// TIA Portal V20 export
DATA_BLOCK "ALARM TABLE"   // DB2025
{ S7_Optimized_Access := 'FALSE' }
// stored: AutoNumber false
   VAR
      TAB_01 : Struct
         CNT01 : Int;
         DBX2_0 : Bool;   // 3;AI;Temperatura Apa in Bazin Pompare - Minim Minim;DI;W2;6;O
         DBX2_1 : Bool;   // 3;AI;Temperatura Apa in Bazin Pompare - Minim;DI;W1;6;O
         DBX2_2 : Bool;   // 3;AI;Temperatura Apa in Bazin Pompare - Maxim;DI;A1;6;O
         DBX2_3 : Bool;   // 3;AI;Temperatura Apa in Bazin Pompare - Maxim Maxim;DI;A2;6;O
         DBX2_4 : Bool;   // 3;AI;Temperatura Apa in Bazin Pompare - Senzor Defect;DI;A2;6;M
         DBX2_5 : Bool;   // 3;AI;Temperatura EtilenGlicol Intrare in Racitor - Minim Minim;DI;W1;6;O
         DBX2_6 : Bool;   // 3;AI;Temperatura EtilenGlicol Intrare in Racitor - Minim;DI;W1;6;O
         DBX2_7 : Bool;   // 3;AI;Temperatura EtilenGlicol Intrare in Racitor - Maxim;DI;W1;6;O
         DBX3_0 : Bool;   // 3;AI;Temperatura EtilenGlicol Intrare in Racitor - Maxim Maxim;DI;A1;6;O
         DBX3_1 : Bool;   // 3;AI;Temperatura EtilenGlicol Intrare in Racit. - Senzor Defect;DI;A2;6;M
         DBX3_2 : Bool;   // 3;AI;Temperatura EtilenGlicol Iesire din Racitor - Minim Minim;DI;W1;6;O
         DBX3_3 : Bool;   // 3;AI;Temperatura EtilenGlicol Iesire din Racitor - Minim;DI;W1;6;O
         DBX3_4 : Bool;   // 3;AI;Temperatura EtilenGlicol Iesire din Racitor - Maxim;DI;W1;6;O
         DBX3_5 : Bool;   // 3;AI;Temperatura EtilenGlicol Iesire din Racitor - Maxim Maxim;DI;A1;6;O
         DBX3_6 : Bool;   // 3;AI;Temperatura EtilenGlicol Iesire din Racit. - Senzor Defect;DI;A2;6;M
         DBX3_7 : Bool;   // 3;AI;Temperatura Apa la Iesire din Racitor - Minim Minim;DI;W2;6;O
         DBX4_0 : Bool;   // 3;AI;Temperatura Apa la Iesire din Racitor - Minim;DI;W1;6;O
         DBX4_1 : Bool;   // 3;AI;Temperatura Apa la Iesire din Racitor - Maxim;DI;W2;6;O
         DBX4_2 : Bool;   // 3;AI;Temperatura Apa la Iesire din Racitor - Maxim Maxim;DI;W2;6;O
         DBX4_3 : Bool;   // 3;AI;Temperatura Apa la Iesire din Racitor - Senzor Defect;DI;A2;6;M
         DBX4_4 : Bool;   // 3;AI;Temperatura Apa Alimentare Linia Calire - Minim Minim;DI;A2;3;O
         DBX4_5 : Bool;   // 3;AI;Temperatura Apa Alimentare Linia Calire - Minim;DI;A1;3;M;O
         DBX4_6 : Bool;   // 3;AI;Temperatura Apa Alimentare Linia Calire - Maxim;DI;A1;3;O
         DBX4_7 : Bool;   // 3;AI;Temperatura Apa Alimentare Linia Calire - Maxim Maxim;DI;A2;3;O
         DBX5_0 : Bool;   // 3;AI;Temperatura Apa Alimentare Linia Calire - Senzor Defect;DI;A2;3;M
         DBX5_1 : Bool;   // 3;AI;Temperatura Apa Alimentare Turnuri Racire - Minim Minim;DI;W2;6;O
         DBX5_2 : Bool;   // 3;AI;Temperatura Apa Alimentare Turnuri Racire - Minim;DI;W1;6;O
         DBX5_3 : Bool;   // 3;AI;Temperatura Apa Alimentare Turnuri Racire - Maxim;DI;A1;6;O
         DBX5_4 : Bool;   // 3;AI;Temperatura Apa Alimentare Turnuri Racire - Maxim Maxim;DI;A1;6;O
         DBX5_5 : Bool;   // 3;AI;Temperatura Apa Alimentare Turnuri Racire - Senzor Defect;DI;A2;6;M
         DBX5_6 : Bool;   // 3;AI;Temparatura Apa in Vas Intermediar - Minim Minim;DI;W1;6;O
         DBX5_7 : Bool;   // 3;AI;Temparatura Apa in Vas Intermediar - Minim;DI;W1;6;O
         DBX6_0 : Bool;   // 3;AI;Temparatura Apa in Vas Intermediar - Maxim;DI;A1;6;O
         DBX6_1 : Bool;   // 3;AI;Temparatura Apa in Vas Intermediar - Maxim Maxim;DI;A1;6;O
         DBX6_2 : Bool;   // 3;AI;Temparatura Apa in Vas Intermediar - Senzor Defect;DI;A2;6;M
         DBX6_3 : Bool;   // 3;AI;Presiune Apa Alimentare Linia Calire - Minim Minim;DI;A2;8;O
         DBX6_4 : Bool;   // 3;AI;Presiune Apa Alimentare Linia Calire - Minim;DI;A1;8;O
         DBX6_5 : Bool;   // 3;AI;Presiune Apa Alimentare Linia Calire - Maxim;DI;A1;8;O
         DBX6_6 : Bool;   // 3;AI;Presiune Apa Alimentare Linia Calire - Maxim Maxim;DI;A2;8;O
         DBX6_7 : Bool;   // 3;AI;Presiune Apa Alimentare Linia Calire - Senzor Defect;DI;A2;8;M
         DBX7_0 : Bool;   // 3;AI;Nivel Apa in Bazin Pompare - Minim Minim;DI;A2;6;O;K
         DBX7_1 : Bool;   // 3;AI;Nivel Apa in Bazin Pompare - Minim;DI;A1;6;O
         DBX7_2 : Bool;   // 3;AI;Nivel Apa in Bazin Pompare - Maxim;DI;A1;6;O;K
         DBX7_3 : Bool;   // 3;AI;Nivel Apa in Bazin Pompare - Maxim Maxim;DI;A2;6;O;K
         DBX7_4 : Bool;   // 3;AI;Nivel Apa in Bazin Pompare - Senzor Defect;DI;A2;6;M
         DBX7_5 : Bool;   // 3;AI;Nivel Apa in Basa Generala - Minim Minim;DI;A2;6;O;K
         DBX7_6 : Bool;   // 3;AI;Nivel Apa in Basa Generala - Minim;DI;A1;6;O
         DBX7_7 : Bool;   // 3;AI;Nivel Apa in Basa Generala - Maxim;DI;A1;6;O
         DBX8_0 : Bool;   // 3;AI;Nivel Apa in Basa Generala - Maxim Maxim;DI;A2;6;O
         DBX8_1 : Bool;   // 3;AI;Nivel Apa in Basa Generala - Senzor Defect;DI;A1;6;M;K
         DBX8_2 : Bool;
         DBX8_3 : Bool;
         DBX8_4 : Bool;
         DBX8_5 : Bool;
         DBX8_6 : Bool;
         DBX8_7 : Bool;
         DBX9_0 : Bool;
         DBX9_1 : Bool;
         DBX9_2 : Bool;
         DBX9_3 : Bool;
         DBX9_4 : Bool;
         DBX9_5 : Bool;
         DBX9_6 : Bool;
         DBX9_7 : Bool;
         DBX10_0 : Bool;
         DBX10_1 : Bool;
         DBX10_2 : Bool;
         DBX10_3 : Bool;
         DBX10_4 : Bool;
         DBX10_5 : Bool;
         DBX10_6 : Bool;
         DBX10_7 : Bool;
         DBX11_0 : Bool;
         DBX11_1 : Bool;
         DBX11_2 : Bool;
         DBX11_3 : Bool;
         DBX11_4 : Bool;
         DBX11_5 : Bool;
         DBX11_6 : Bool;
         DBX11_7 : Bool;
         DBX12_0 : Bool;   // 3;AI;Temperatura Teava (pirometru dupa Sutton) - Minim Minim;DI;A2;20;O
         DBX12_1 : Bool;   // 3;AI;Temperatura Teava (pirometru dupa Sutton) - Minim;DI;A1;20;O
         DBX12_2 : Bool;   // 3;AI;Temperatura Teava (pirometru dupa Sutton) - Maxim;DI;A1;20;O
         DBX12_3 : Bool;   // 3;AI;Temperatura Teava (pirometru dupa Sutton) - Maxim Maxim;DI;A2;20;O
         DBX12_4 : Bool;   // 3;AI;Temperatura Teava (pirometru dupa Sutton) - Senzor Defect;DI;A2;20;M
         DBX12_5 : Bool;   // 3;AI;Temperatura Teava (pir. intr. cupt. revenire) - Minim Minim;DI;A1;20;O
         DBX12_6 : Bool;   // 3;AI;Temperatura Teava (pir. intr. cupt. revenire) - Minim;DI;A1;20;O
         DBX12_7 : Bool;   // 3;AI;Temperatura Teava (pir. intr. cupt. revenire) - Maxim;DI;A1;20;O
         DBX13_0 : Bool;   // 3;AI;Temperatura Teava (pir. intr. cupt. revenire) - Maxim Maxim;DI;A2;20;O
         DBX13_1 : Bool;   // 3;AI;Temperatura Teava (pir. intr. cupt. revenire) - Senzor Def.;DI;A2;20;M
         DBX13_2 : Bool;   // 3;AI;Low Low Apa Redox;DI;A2;20;M;O
         DBX13_3 : Bool;
         DBX13_4 : Bool;
         DBX13_5 : Bool;
         DBX13_6 : Bool;
         DBX13_7 : Bool;
         DBX14_0 : Bool;
         DBX14_1 : Bool;
         DBX14_2 : Bool;
         DBX14_3 : Bool;
         DBX14_4 : Bool;
         DBX14_5 : Bool;
         DBX14_6 : Bool;
         DBX14_7 : Bool;
         DBX15_0 : Bool;
         DBX15_1 : Bool;
         DBX15_2 : Bool;
         DBX15_3 : Bool;
         DBX15_4 : Bool;
         DBX15_5 : Bool;
         DBX15_6 : Bool;
         DBX15_7 : Bool;
         DBX16_0 : Bool;
         DBX16_1 : Bool;
         DBX16_2 : Bool;
         DBX16_3 : Bool;
         DBX16_4 : Bool;
         DBX16_5 : Bool;
         DBX16_6 : Bool;
         DBX16_7 : Bool;
         DBX17_0 : Bool;   // 3;AI;Lipsa presiune destunderizator;DI;A2;7;O
         DBX17_1 : Bool;   // 3;AI;Nivel Apa in Bazin Pompare - Minim;DI;A1;7;O
         DBX17_2 : Bool;
         DBX17_3 : Bool;
         DBX17_4 : Bool;
         DBX17_5 : Bool;
         DBX17_6 : Bool;   // 5;ROLLS T6;Problema pirometru intrare cuptor;DI;A1;16;M;O
         DBX17_7 : Bool;   // 4;FIERASTRAU KASTO;Pat racire - Zona Kasto pachete diferite;TK;W2;11;O
         DBX18_0 : Bool;
         DBX18_1 : Bool;
         DBX18_2 : Bool;
         DBX18_3 : Bool;
         DBX18_4 : Bool;
         DBX18_5 : Bool;
         DBX18_6 : Bool;
         DBX18_7 : Bool;
         DBX19_0 : Bool;
         DBX19_1 : Bool;
         DBX19_2 : Bool;
         DBX19_3 : Bool;
         DBX19_4 : Bool;
         DBX19_5 : Bool;
         DBX19_6 : Bool;
         DBX19_7 : Bool;
         DBX20_0 : Bool;
         DBX20_1 : Bool;
         DBX20_2 : Bool;
         DBX20_3 : Bool;
         DBX20_4 : Bool;
         DBX20_5 : Bool;
         DBX20_6 : Bool;
         DBX20_7 : Bool;
         DBX21_0 : Bool;
         DBX21_1 : Bool;
         DBX21_2 : Bool;
         DBX21_3 : Bool;
         DBX21_4 : Bool;
         DBX21_5 : Bool;
         DBX21_6 : Bool;
         DBX21_7 : Bool;
         DBX22_0 : Bool;
         DBX22_1 : Bool;
         DBX22_2 : Bool;
         DBX22_3 : Bool;
         DBX22_4 : Bool;
         DBX22_5 : Bool;
         DBX22_6 : Bool;
         DBX22_7 : Bool;
         DBX23_0 : Bool;
         DBX23_1 : Bool;
         DBX23_2 : Bool;
         DBX23_3 : Bool;
         DBX23_4 : Bool;
         DBX23_5 : Bool;
         DBX23_6 : Bool;
         DBX23_7 : Bool;
         DBX24_0 : Bool;
         DBX24_1 : Bool;
         DBX24_2 : Bool;
         DBX24_3 : Bool;
         DBX24_4 : Bool;
         DBX24_5 : Bool;
         DBX24_6 : Bool;
         DBX24_7 : Bool;
         DBX25_0 : Bool;
         DBX25_1 : Bool;
         DBX25_2 : Bool;
         DBX25_3 : Bool;
         DBX25_4 : Bool;
         DBX25_5 : Bool;
         DBX25_6 : Bool;
         DBX25_7 : Bool;
         DBX26_0 : Bool;
         DBX26_1 : Bool;
         DBX26_2 : Bool;
         DBX26_3 : Bool;
         DBX26_4 : Bool;
         DBX26_5 : Bool;
         DBX26_6 : Bool;
         DBX26_7 : Bool;
         DBX27_0 : Bool;
         DBX27_1 : Bool;
         DBX27_2 : Bool;
         DBX27_3 : Bool;
         DBX27_4 : Bool;
         DBX27_5 : Bool;
         DBX27_6 : Bool;
         DBX27_7 : Bool;
         DBX28_0 : Bool;
         DBX28_1 : Bool;
         DBX28_2 : Bool;
         DBX28_3 : Bool;
         DBX28_4 : Bool;
         DBX28_5 : Bool;
         DBX28_6 : Bool;
         DBX28_7 : Bool;
         DBX29_0 : Bool;
         DBX29_1 : Bool;
         DBX29_2 : Bool;
         DBX29_3 : Bool;
         DBX29_4 : Bool;
         DBX29_5 : Bool;
         DBX29_6 : Bool;
         DBX29_7 : Bool;
         DBX30_0 : Bool;
         DBX30_1 : Bool;
         DBX30_2 : Bool;
         DBX30_3 : Bool;
         DBX30_4 : Bool;
         DBX30_5 : Bool;
         DBX30_6 : Bool;
         DBX30_7 : Bool;
         DBX31_0 : Bool;
         DBX31_1 : Bool;
         DBX31_2 : Bool;
         DBX31_3 : Bool;
         DBX31_4 : Bool;
         DBX31_5 : Bool;
         DBX31_6 : Bool;
         DBX31_7 : Bool;
         DBX32_0 : Bool;   // 1;Gen;Z1:Sistem Oprire de Urgenta T1-A - Declansat;EM;A3;1;M;O;K
         DBX32_1 : Bool;   // 1;Gen;Z2:Sistem Oprire de Urgenta T1-C - Declansat;EM;A3;1;M;O;K
         DBX32_2 : Bool;   // 1;Gen;Z3:Sistem Oprire de Urgenta Apa - Declansat;EM;A3;6;M;O;K
         DBX32_3 : Bool;   // 1;Gen;Z4:Sistem Oprire de Urgenta T3,T4 - Declansat;EM;A3;10;M;O;K
         DBX32_4 : Bool;   // 1;Gen;Z5:Sistem Oprire de Urgenta T5-T6 - Declansat;EM;A3;14;M;O;K
         DBX32_5 : Bool;   // 1;Gen;Z6:Sistem Oprire de Urgenta T1-D - Declansat;EM;A3;16;M;O;K
         DBX32_6 : Bool;   // 1;Gen;Z7:Sistem Oprire de Urgenta T7 - Declansat;EM;A3;21;M;O;K
         DBX32_7 : Bool;   // 1;Gen;Z8:Sistem Oprire de Urgenta T7-A,T7-B,T7-C - Declansat;EM;A3;23;M;O;K
         DBX33_0 : Bool;   // 1;Gen;Lipsa Tensiune Alimentare Intrari Digitale PLC;DI;A1;6;M;K
         DBX33_1 : Bool;   // 1;Gen;Lipsa Tensiune Alimentare Iesiri Digitale PLC;DI;A1;6;M;K
         DBX33_2 : Bool;   // 1;Gen;Lipsa Tensiune Alimentare (220V pt. module ET);DI;A1;6;M;K
         DBX33_3 : Bool;   // 1;Gen;Lipsa Tensiune Alimentare pt. modulele ET-TF1;DI;A1;6;M;K
         DBX33_4 : Bool;   // 1;Gen;Lipsa Tensiune Alimentare pt. modulele ET-TF2;DI;A1;20;M;K
         DBX33_5 : Bool;   // 1;Gen;Lipsa Tensiune Alimentare pt. modulele ET-TF3;DI;A1;6;M;K
         DBX33_6 : Bool;   // 1;Gen;Lipsa Tensiune Alimentare pt. modulele ET-TF4;DI;A1;6;M;K
         DBX33_7 : Bool;   // 1;Gen;Lipsa Tensiune Alimentare pt. modulele ET-LM1;DI;A1;6;M;K
         DBX34_0 : Bool;   // 1;Gen;Lipsa Tensiune Alimentare pt. modulele ET-LM2;DI;A1;6;M;K
         DBX34_1 : Bool;   // 1;Gen;Lipsa Tensiune Alimentare pt. modulele ET-LM4;DI;A1;13;M;K
         DBX34_2 : Bool;   // 1;Gen;Lipsa Tensiune Alimentare pt. modulele ET-LM5;DI;A1;20;M;K
         DBX34_3 : Bool;   // 1;Gen;Lipsa Tensiune Alimentare pt. modulele ET-LM6;DI;A1;27;M;K
         DBX34_4 : Bool;   // 1;Gen;Lipsa Tensiune Alimentare pt. modulele ET-LM7;DI;A1;6;M;K
         DBX34_5 : Bool;   // 1;Gen;Z1:Teava mai lunga de 14m pe T1-A Incarcare imposibila;DI;A3;1;M;O;K
         DBX34_6 : Bool;   // 1;Gen;Lipsa Tensiune Alimentare UPS;DI;W2;6;M
         DBX34_7 : Bool;   // 1;Gen;UPS not OK;DI;W2;6;M
         DBX35_0 : Bool;   // 1;Gen;Lipsa Tensiune Alimentare pt. Electrovalvole (PLC);DI;A1;6;M;K
         DBX35_1 : Bool;   // 1;Gen;Lipsa Tensiune Alimentare pt. Electrovalvole (LM1);DI;A1;6;M;K
         DBX35_2 : Bool;   // 1;Gen;Lipsa Tensiune Alimentare pt. Electrovalvole (LM2);DI;A1;6;M;K
         DBX35_3 : Bool;   // 1;Gen;Lipsa Tensiune Alimentare pt. Electrovalvole (LM4);DI;A1;6;M;K
         DBX35_4 : Bool;   // 1;Gen;Lipsa Tensiune Alimentare pt. Electrovalvole (LM5);DI;A1;6;M;K
         DBX35_5 : Bool;   // 1;Gen;Lipsa Tensiune Alimentare pt. Electrovalvole (LM6);DI;A1;6;M;K
         DBX35_6 : Bool;   // 1;Gen;Lipsa Tensiune Alimentare pt. Electrovalvole (LM7);DI;A1;6;M;K
         DBX35_7 : Bool;   // 1;Gen;Lipsa Tensiune Alimentare pt. Electrovalvole (ET-TF1);DI;A1;6;M;K
         DBX36_0 : Bool;   // 1;Gen;Lipsa Tensiune Alimentare Senzori (LM1);DI;A1;6;M;K
         DBX36_1 : Bool;   // 1;Gen;Lipsa Tensiune Alimentare Senzori(LM2);DI;A1;6;M;K
         DBX36_2 : Bool;   // 1;Gen;Lipsa Tensiune Alimentare Senzori(LM4);DI;A1;6;M;K
         DBX36_3 : Bool;   // 1;Gen;Lipsa Tensiune Alimentare Senzori(LM5);DI;A1;6;M;K
         DBX36_4 : Bool;   // 1;Gen;Lipsa Tensiune Alimentare Senzori(LM6);DI;A1;6;M;K
         DBX36_5 : Bool;   // 1;LM1;Lipsa Tensiune Alimentare Intrari Digitale (LM1);DI;A1;13;M;K
         DBX36_6 : Bool;   // 1;LM1;Lipsa Tensiune Alimentare Iesiri Digitale (LM1);DI;A1;13;M;K
         DBX36_7 : Bool;   // 1;LM1;Lipsa Tensiune Alimentare Modul FM350 (LM1);DI;A1;13;M;K
         DBX37_0 : Bool;
         DBX37_1 : Bool;
         DBX37_2 : Bool;
         DBX37_3 : Bool;   // 1;LM2;Lipsa Tensiune Alimentare Intrari Digitale (LM2);DI;A1;6;M;K
         DBX37_4 : Bool;   // 1;LM2;Lipsa Tensiune Alimentare Iesiri Digitale (LM2);DI;A1;6;M;K
         DBX37_5 : Bool;   // 1;LM2;Lipsa Tensiune Alimentare Modul FM350 (LM2);DI;A1;6;M;K
         DBX37_6 : Bool;
         DBX37_7 : Bool;
         DBX38_0 : Bool;
         DBX38_1 : Bool;   // 1;LM4;Lipsa Tensiune Alimentare Intrari Digitale (LM4);DI;A1;6;M;K
         DBX38_2 : Bool;   // 1;LM4;Lipsa Tensiune Alimentare Iesiri Digitale (LM4);DI;A1;6;M;K
         DBX38_3 : Bool;   // 1;PLC;TimeOut Comunicatie cu PLC-ul de la Cuptorul de Calire;DI;A1;3;M;O;K
         DBX38_4 : Bool;   // 6;PLC;TimeOut Comunicatie cu PLC-ul de la Cuptorul de Revenire;DI;A1;17;M;O;K
         DBX38_5 : Bool;   // 8;PLC;TimeOut Comunicatie cu PLC-ul de la Indreptare Tevi ;DI;A1;22;M;O;K
         DBX38_6 : Bool;
         DBX38_7 : Bool;   // 1;LM5;Lipsa Tensiune Alimentare Intrari Digitale (LM5);DI;A1;20;M;K
         DBX39_0 : Bool;   // 1;LM5;Lipsa Tensiune Alimentare Iesiri Digitale (LM5);DI;A1;20;M;K
         DBX39_1 : Bool;   // 1;LM5;Lipsa Tensiune Alimentare Modul FM350 (LM5);DI;A1;20;M;K
         DBX39_2 : Bool;
         DBX39_3 : Bool;
         DBX39_4 : Bool;
         DBX39_5 : Bool;   // 1;LM6;Lipsa Tensiune Alimentare Intrari Digitale (LM6);DI;A1;27;M;K
         DBX39_6 : Bool;   // 1;LM6;Lipsa Tensiune Alimentare Iesiri Digitale (LM6);DI;A1;27;M;K
         DBX39_7 : Bool;   // 1;LM6;Lipsa Tensiune Alimentare Modul FM350 (LM6);DI;A1;27;M;K
         DBX40_0 : Bool;
         DBX40_1 : Bool;
         DBX40_2 : Bool;
         DBX40_3 : Bool;   // 1;LM7;Lipsa Tensiune Alimentare Intrari Digitale (LM7);DI;A1;27;M;K
         DBX40_4 : Bool;   // 1;LM7;Lipsa Tensiune Alimentare Iesiri Digitale (LM7);DI;A1;27;M;K
         DBX40_5 : Bool;   // 1;LM7;Lipsa Tensiune Alimentare Senzori (LM6);DI;A1;27;M;K
         DBX40_6 : Bool;
         DBX40_7 : Bool;
         DBX41_0 : Bool;   // 1;TF1;Lipsa Tensiune Alimentare Intrari Digitale (TF1);DI;A1;6;M;K
         DBX41_1 : Bool;   // 1;TF1;Lipsa Tensiune Alimentare Iesiri Digitale (TF1);DI;A1;6;M;K
         DBX41_2 : Bool;   // 1;TF1;Lipsa Tensiune Alimentare 380V (TF1);DI;A1;6;M;K
         DBX41_3 : Bool;   // 1;TF1;Lipsa Tensiune Alimentare 220V (TF1);DI;A1;6;M;K
         DBX41_4 : Bool;   // 1;TF1;Disjunctor Termic 220V (TF1) - Declansat;DI;A1;6;M;K
         DBX41_5 : Bool;
         DBX41_6 : Bool;
         DBX41_7 : Bool;   // 1;TF2;Lipsa Tensiune Alimentare Intrari Digitale (TF2);DI;A1;20;M;K
         DBX42_0 : Bool;   // 1;TF2;Lipsa Tensiune Alimentare Iesiri Digitale (TF2);DI;A1;20;M;K
         DBX42_1 : Bool;
         DBX42_2 : Bool;
         DBX42_3 : Bool;   // 1;TF3;Lipsa Tensiune Alimentare Intrari Digitale (TF3);DI;A1;27;M;K
         DBX42_4 : Bool;   // 1;TF3;Lipsa Tensiune Alimentare Iesiri Digitale (TF3);DI;A1;27;M;K
         DBX42_5 : Bool;   // 1;TF3;Lipsa Tensiune Alimentare 380V (TF3);DI;A1;27;M;K
         DBX42_6 : Bool;   // 1;TF3;Lipsa Tensiune Alimentare 220V (TF3);DI;A1;27;M;K
         DBX42_7 : Bool;   // 1;TF3;Disjunctor Termic 220V (TF3) - Declansat;DI;A1;27;M;K
         DBX43_0 : Bool;
         DBX43_1 : Bool;
         DBX43_2 : Bool;   // 1;TF4;Lipsa Tensiune Alimentare Intrari Digitale (TF4);DI;A1;6;M;K
         DBX43_3 : Bool;   // 1;TF4;Lipsa Tensiune Alimentare Senzori (TF4);DI;A1;6;M;K
         DBX43_4 : Bool;
         DBX43_5 : Bool;
         DBX43_6 : Bool;   // 4;Gen;Z4:Sistem Oprire de Urgenta Role RC02 T4 - Declansat;EM;A3;10;M;O;K
         DBX43_7 : Bool;   // 10;Gen;Z27:Sistem Oprire de Urgenta T10 EH01 - Declansat;EM;A3;28;M;O;K
         DBX44_0 : Bool;   // 10;Gen;Z27:Sistem Oprire de Urgenta T10 EH10 - Declansat;EM;A3;28;M;O;K
         DBX44_1 : Bool;   // 10;Gen;Z27:Sistem Oprire de Urgenta T10 EH11 - Declansat;EM;A3;28;M;O;K
         DBX44_2 : Bool;   // 5;Gen;Z15:Sistem Oprire de Urgenta T6 Kasto EH10 - Declansat;EM;A3;15;M;O;K
         DBX44_3 : Bool;   // 9;Gen;Z25:Sistem Oprire de Urgenta T7-C Kasto EH10 - Declansat;EM;A3;25;M;O;K
         DBX44_4 : Bool;
         DBX44_5 : Bool;
         DBX44_6 : Bool;
         DBX44_7 : Bool;
         DBX45_0 : Bool;   // 10;EGH01;Lipsa Tensiune Alimentare 380V (EGH01);DI;A3;28;M;K
         DBX45_1 : Bool;   // 10;EGH01;Lipsa Tensiune Alimentare 230V (EGH01);DI;A2;28;M;K
         DBX45_2 : Bool;   // 10;EGH01;Lipsa Tensiune Alimentare 230V (EGH01);DI;A2;28;M;K
         DBX45_3 : Bool;   // 10;EGH01;Lipsa Tensiune Alimentare 110V (EGH01);DI;A2;28;M;K
         DBX45_4 : Bool;   // 10;EGH01;Lipsa Tensiune Alimentare 24V Convertizoare (EGH01);DI;A2;28;M;K
         DBX45_5 : Bool;   // 10;EGH01;Lipsa Tensiune Alimentare Electrovalve (EGH01);DI;A2;28;M;K
         DBX45_6 : Bool;   // 10;EGH01;Lipsa Tensiune Alimentare MPP1 (EGH01);DI;A2;28;M;K
         DBX45_7 : Bool;   // 10;EGH01;Lipsa Tensiune Alimentare MPP2 (EGH01);DI;A2;28;M;K
         DBX46_0 : Bool;   // 10;EGH01;Lipsa Tensiune Alimentare Kasto 1(EGH01);DI;A3;28;M;K
         DBX46_1 : Bool;   // 10;EH01;Lipsa Tensiune Alimentare ET(EH01);DI;A2;28;M;K
         DBX46_2 : Bool;   // 10;EH01;Lipsa Tensiune Alimentare Intrari Digitale(EH01);DI;A2;28;M;K
         DBX46_3 : Bool;   // 10;EH01;Lipsa Tensiune Alimentare Iesiri Digitale(EH01);DI;A2;28;M;K
         DBX46_4 : Bool;   // 10;EH01;Lipsa Tensiune Alimentare Dispozitive Aux(EH01);DI;A1;28;M;K
         DBX46_5 : Bool;   // 10;EH01;Lipsa Tensiune Alimentare Encodere(EH01);DI;A3;28;M;K
         DBX46_6 : Bool;   // 0;EH01;Disjunctor Alimentare ET - Declansat(EH01);DI;A2;28;M;K
         DBX46_7 : Bool;
         DBX47_0 : Bool;   // 10;ROLLS T10-1;Lipsa Tensiune de Comanda C.Role T10-1;DI;A1;28;M;K
         DBX47_1 : Bool;   // 10;ROLLS T10-1;Probleme Fuzibil C.Role T10-1;DI;A1;28;M;K
         DBX47_2 : Bool;   // 10;ROLLS T10-1;Disj. Termic Mot. C.Role T10-1 - Declansat;DI;A1;28;M;K
         DBX47_3 : Bool;   // 10;ROLLS T10-1;Fuzibil Neinserat C.Role T10-1;DI;A1;28;M;K
         DBX47_4 : Bool;   // 10;ROLLS T10-1;Inverter Mot. C.Role T10-1 - Avarie;DI;A1;28;M;O;K
         DBX47_5 : Bool;   // 10;ROLLS T10-1;Role T10-1 TimeOut Pozitionare Teava;SQ;A1;28;O
         DBX47_6 : Bool;   // 10;ROLLS T10-1;TimeOut Rotire Role C.Role T10-1;DI;A1;28;M;O;K
         DBX47_7 : Bool;   // 10;ROLLS T10-1;TimeOut Cuplare/Decuplare Vent.Mot.C.RoleT10-1;DI;A1;28;M;O
         DBX48_0 : Bool;   // 10;ROLLS T10-1;Disjunctor Th. AlimVent.Mot.C.Role T10-1 Declansat;DI;A1;28;M
         DBX48_1 : Bool;
         DBX48_2 : Bool;
         DBX48_3 : Bool;
         DBX48_4 : Bool;
         DBX48_5 : Bool;
         DBX48_6 : Bool;
         DBX48_7 : Bool;
         DBX49_0 : Bool;
         DBX49_1 : Bool;
         DBX49_2 : Bool;
         DBX49_3 : Bool;
         DBX49_4 : Bool;
         DBX49_5 : Bool;
         DBX49_6 : Bool;   // 3;T3 SERVOVALVE;Lipsa Tensiune Alimentare Servovalva T3;DI;A1;8;M;K
         DBX49_7 : Bool;   // 3;T3 SERVOVALVE;Disjunctor Termic Servovalva - Declansat;DI;A1;8;M;K
         DBX50_0 : Bool;   // 3;PUMP 1;Disjunctor Termic Pompa Apa Nr.1 - Declansat;DI;A1;6;M
         DBX50_1 : Bool;   // 3;PUMP 2;Disjunctor Termic Pompa Apa Nr.2 - Declansat;DI;A1;6;M
         DBX50_2 : Bool;   // 3;PUMP 3;Disjunctor Termic Pompa Apa Nr.3 - Declansat;DI;A1;6;M
         DBX50_3 : Bool;   // 3;PUMP 4;Disjunctor Termic Pompa Apa Nr.4 - Declansat;DI;A1;6;M
         DBX50_4 : Bool;   // 3;PUMP 5;Disjunctor Termic Pompa Apa Nr.5 - Declansat;DI;A1;6;M
         DBX50_5 : Bool;   // 3;PUMP 6;Disjunctor Termic Pompa Apa Nr.6 - Declansat;DI;A1;6;M
         DBX50_6 : Bool;   // 3;PUMP 7;Disjunctor Termic Pompa Apa Nr.7 - Declansat;DI;A1;6;M
         DBX50_7 : Bool;   // 3;PUMP 8;Disjunctor Termic Pompa Apa Nr.8 - Declansat;DI;A1;6;M
         DBX51_0 : Bool;   // 3;PUMP 9;Disjunctor Termic Pompa Apa Nr.9 - Declansat;DI;A1;6;M
         DBX51_1 : Bool;   // 3;PUMP 10;Disjunctor Termic Pompa Apa Nr.10 - Declansat;DI;A1;6;M
         DBX51_2 : Bool;   // 3;PUMP 11;Disjunctor Termic Pompa Apa Nr.11 - Declansat;DI;A1;6;M
         DBX51_3 : Bool;   // 3;TE1;Disjunctor Termic Transportator Elicoidal Nr.1-Declansat;DI;A1;6;M
         DBX51_4 : Bool;   // 3;TE2;Disjunctor Termic Transportator Elicoidal Nr.2-Declansat;DI;A1;6;M
         DBX51_5 : Bool;   // 3;VE1;Disjunctor Termic Ventilator Turn Racire Nr.1-Declansat;DI;A1;6;M
         DBX51_6 : Bool;   // 3;VE2;Disjunctor Termic Ventilator Turn Racire Nr.2-Declansat;DI;A1;6;M
         DBX51_7 : Bool;   // 3;T3 FILTER;Interupator Termic Filtru T3 - Declansat;DI;A1;8;M
         DBX52_0 : Bool;   // 3;PUMP 1;Lipsa Apa in Pompa Apa Nr.1 (senzor curgere);DI;A1;6;M;O
         DBX52_1 : Bool;   // 3;PUMP 2;Lipsa Apa in Pompa Apa Nr.2 (senzor curgere);DI;A1;6;M;O
         DBX52_2 : Bool;   // 3;PUMP 3;Lipsa Apa in Pompa Apa Nr.3 (senzor curgere);DI;A1;6;M;O
         DBX52_3 : Bool;   // 3;PUMP 4;Lipsa Apa in Pompa Apa Nr.4 (senzor curgere);DI;A1;6;M;O
         DBX52_4 : Bool;   // 3;PUMP 5;Lipsa Apa in Pompa Apa Nr.5 (senzor curgere);DI;A1;6;M;O
         DBX52_5 : Bool;   // 3;PUMP 6;Lipsa Apa in Pompa Apa Nr.5R (senzor curgere);DI;A1;6;M;O
         DBX52_6 : Bool;   // 3;PUMP 7;Lipsa Apa in Pompa Apa Nr.7 (senzor curgere);DI;A1;6;M;O
         DBX52_7 : Bool;   // 3;PUMP 8;Lipsa Apa in Pompa Apa Nr.8 (senzor curgere);DI;A1;6;M;O
         DBX53_0 : Bool;   // 3;T3 FILTER;Lipsa Tensiune Alimentare Filtru T3;DI;A1;8;M;K
         DBX53_1 : Bool;   // 3;PUMP 10;Lipsa Apa in Pompa Apa Nr.10 (senzor curgere);DI;A1;6;M;O
         DBX53_2 : Bool;   // 3;BASIN;Lipsa Apa in Bazinul de Pompare;DI;A1;6;O
         DBX53_3 : Bool;   // 3;PUMP 11;Nivel Apa in Casa Pompelor - Minim;DI;A1;6;O
         DBX53_4 : Bool;   // 3;PUMP 11;Nivel Apa in Casa Pompelor - Maxim;DI;A2;6;O;K
         DBX53_5 : Bool;   // 3;BASIN;Nivel Apa in Bazinul de Pompare - Maxim;DI;A2;6;O;K
         DBX53_6 : Bool;   // 3;VESSEL;Nivel Apa in Vasul Intermediar - Minim;DI;A2;6;O;K
         DBX53_7 : Bool;   // 3;T3 FILTER/BEAM;Lipsa Tensiune de Comanda Filtru T3 si Grinda;DI;A2;8;M;K
         DBX54_0 : Bool;   // 3;SCALE;Nivel Apa in Bazinul Tunder - Maxim;DI;A2;6;O;K
         DBX54_1 : Bool;   // 3;SUP;Presiune Apa Scazuta pe Linia de Calire;DI;A1;6;O;K
         DBX54_2 : Bool;   // 3;TOWER;Presiune Apa Scazuta pe Linia de Racire Turnuri;DI;A1;6;O;K
         DBX54_3 : Bool;   // 3;SCP;Temperatura Apa din Schimbatorul de Caldura - Depasita;DI;A2;6;M
         DBX54_4 : Bool;   // 3;BASIN;Temperatura Apa din Bazinul de Pompare - Depasita;DI;A2;6;M;O;K
         DBX54_5 : Bool;   // 3;BASIN;Temperatura Apa din Bazinul de Pompare - Scazuta;DI;A1;6;M;O
         DBX54_6 : Bool;   // 3;BASIN;Avarie Schimbator Caldura (cu EtilenGlicol);DI;A1;6;M;O
         DBX54_7 : Bool;   // 3;DCS;Avarie Sistem DCS;DI;A3;6;M;O;K
         DBX55_0 : Bool;   // 3;F;Avarie Filtru cu Autocuratire;DI;W3;6;O
         DBX55_1 : Bool;   // 3;PUMP 1;TimeOut Cuplare Contactor Pornire Pompa Apa Nr.1;DI;A1;6;M;O;K
         DBX55_2 : Bool;   // 3;PUMP 2;TimeOut Cuplare Contactor Pornire Pompa Apa Nr.2;DI;A1;6;M;O;K
         DBX55_3 : Bool;   // 3;PUMP 3;TimeOut Cuplare Contactor Pornire Pompa Apa Nr.3;DI;A1;6;M;O;K
         DBX55_4 : Bool;   // 3;PUMP 4;TimeOut Cuplare Contactor Pornire Pompa Apa Nr.4;DI;A1;6;M;O;K
         DBX55_5 : Bool;   // 3;PUMP 5;TimeOut Cuplare Contactor Pornire Pompa Apa Nr.5;DI;A1;6;M;O;K
         DBX55_6 : Bool;   // 3;PUMP 5R;TimeOut Cuplare Contactor Pornire Pompa Apa Nr.5R;DI;A1;6;M;O;K
         DBX55_7 : Bool;   // 3;PUMP 7;TimeOut Cuplare Contactor Pornire Pompa Apa Nr.7;DI;A1;6;M;O;K
         DBX56_0 : Bool;   // 3;PUMP 8;TimeOut Cuplare Contactor Pornire Pompa Apa Nr.8;DI;A1;6;M;O;K
         DBX56_1 : Bool;   // 3;PUMP 9;TimeOut Cuplare Contactor Pornire Pompa Apa Nr.9;DI;A1;6;M;O;K
         DBX56_2 : Bool;   // 3;PUMP10;TimeOut Cuplare Contactor Pornire Pompa Apa Nr10;DI;A1;6;M;O;K
         DBX56_3 : Bool;   // 3;PUMP11;TimeOut Cuplare Contactor Pornire Pompa Apa Nr11;DI;A1;6;M;O;K
         DBX56_4 : Bool;   // 3;HELICOIDAL TRANSPORTER 1;TimeOut Transportator Elicoidal Nr.1;DI;A1;6;M;O;K
         DBX56_5 : Bool;   // 3;HELICOIDAL TRANSPORTER 2;TimeOut Transportator Elicoidal Nr.2;DI;A1;6;M;O;K
         DBX56_6 : Bool;   // 3;COOLING TOWER 1;TimeOut Ventilator Turn Racire 1 Viteza Mica;DI;A1;6;M;O;K
         DBX56_7 : Bool;   // 3;COOLING TOWER 1;TimeOut Ventilator Turn Racire 1 Viteza Mare;DI;A1;6;M;O;K
         DBX57_0 : Bool;   // 3;COOLING TOWER 2;TimeOut Ventilator Turn Racire 2 Viteza Mica;DI;A1;6;M;O;K
         DBX57_1 : Bool;   // 3;COOLING TOWER 2;TimeOut Ventilator Turn Racire 2 Viteza Mare;DI;A1;6;M;O;K
         DBX57_2 : Bool;   // 3;T3 FILTER;TimeOut Cuplare/Decuplare Contactor Filtru Inainte;DI;A1;8;M;O;K
         DBX57_3 : Bool;   // 3;T3 FILTER;TimeOut Cuplare/Decuplare Contactor Filtru Inapoi;DI;A1;8;M;O;K
         DBX57_4 : Bool;
         DBX57_5 : Bool;   // 3;T3 SERVOVALVE;Lipsa Tensiune Alimentare Servovalva;DI;A1;8;M;K
         DBX57_6 : Bool;
         DBX57_7 : Bool;
         DBX58_0 : Bool;   // 1;CHAIN T1-A;TimeOut Cuplare Contactor Start Lant T1-A;DI;A1;1;M;O;K
         DBX58_1 : Bool;
         DBX58_2 : Bool;   // 1;CHAIN T1-A;TimeOut Deplasare Lant T1-A in pozitia Pas;DI;A1;1;M;O;K
         DBX58_3 : Bool;   // 1;CHAIN T1-A;Disjunctor Termic Lant T1-A - Declansat;DI;A1;1;M;K
         DBX58_4 : Bool;   // 1;CHAIN T1-A;Sectionator Alimentare Lant T1-A - Decuplat;DI;A1;1;M;K
         DBX58_5 : Bool;   // 1;STOPPER T1-A;Disjunctor Termic Opritor T1-A - Declansat;DI;A1;1;M;K
         DBX58_6 : Bool;   // 1;STOPPER T1-A;Sectionator Alimentare Opritor T1-A - Decuplat;DI;A1;1;M;K
         DBX58_7 : Bool;   // 1;STOPPER T1-A;TimeOut Cuplare Contactor Opritor T1-A;DI;A1;1;M;O;K
         DBX59_0 : Bool;   // 3;T3 FILTER;Lipsa confirmare rotire filtru delta T3;DI;A1;1;M;K
         DBX59_1 : Bool;
         DBX59_2 : Bool;
         DBX59_3 : Bool;
         DBX59_4 : Bool;
         DBX59_5 : Bool;
         DBX59_6 : Bool;
         DBX59_7 : Bool;
         DBX60_0 : Bool;
         DBX60_1 : Bool;
         DBX60_2 : Bool;
         DBX60_3 : Bool;
         DBX60_4 : Bool;
         DBX60_5 : Bool;
         DBX60_6 : Bool;
         DBX60_7 : Bool;
         DBX61_0 : Bool;
         DBX61_1 : Bool;
         DBX61_2 : Bool;
         DBX61_3 : Bool;
         DBX61_4 : Bool;
         DBX61_5 : Bool;
         DBX61_6 : Bool;
         DBX61_7 : Bool;
         DBX62_0 : Bool;   // 1;FLIPPER T1A;Lipsa Tensiune Alimentare Aruncator T1-A;DI;A1;1;M;K
         DBX62_1 : Bool;   // 1;FLIPPER T1A;TimeOut Deplasare Aruncator T1-A in pozitia Sus;DI;A1;1;M;O
         DBX62_2 : Bool;   // 1;FLIPPER T1A;TimeOut Deplasare Aruncator T1-A in pozitia Jos;DI;A1;1;M;O
         DBX62_3 : Bool;   // 1;FLIPPER T1A;Eroare Depozitare Teava pe C.Role T1-A;SQ;A1;1;O
         DBX62_4 : Bool;
         DBX62_5 : Bool;
         DBX62_6 : Bool;
         DBX62_7 : Bool;
         DBX63_0 : Bool;
         DBX63_1 : Bool;
         DBX63_2 : Bool;
         DBX63_3 : Bool;
         DBX63_4 : Bool;
         DBX63_5 : Bool;
         DBX63_6 : Bool;
         DBX63_7 : Bool;
         DBX64_0 : Bool;
         DBX64_1 : Bool;
         DBX64_2 : Bool;
         DBX64_3 : Bool;
         DBX64_4 : Bool;
         DBX64_5 : Bool;
         DBX64_6 : Bool;
         DBX64_7 : Bool;
         DBX65_0 : Bool;
         DBX65_1 : Bool;
         DBX65_2 : Bool;
         DBX65_3 : Bool;
         DBX65_4 : Bool;
         DBX65_5 : Bool;
         DBX65_6 : Bool;
         DBX65_7 : Bool;
         DBX66_0 : Bool;   // 1;ROLLS T1-A;Suma Disjuntoare Termice C.Role T1-A - Declansat;DI;A1;1;M;K
         DBX66_1 : Bool;   // 1;ROLLS T1-A;Sectionator Alim.Inverter C.Role T1-A - Decuplat;DI;A2;1;M;K
         DBX66_2 : Bool;   // 1;ROLLS T1-A;Lipsa Tensiune de Comanda C.Role T1-A;DI;A2;1;M;K
         DBX66_3 : Bool;   // 1;ROLLS T1-A;TimeOut Rotire Role C.Role T1-A;DI;A1;1;M;O;K
         DBX66_4 : Bool;   // 1;ROLLS T1-A;Disj. Termic Rola Nr.1 C.Role T1-A Declansat;DI;W2;1;M
         DBX66_5 : Bool;   // 1;ROLLS T1-A;Disj. Termic Rola Nr.2 C.Role T1-A Declansat;DI;W2;1;M
         DBX66_6 : Bool;   // 1;ROLLS T1-A;Disj. Termic Rola Nr.3 C.Role T1-A Declansat;DI;W2;1;M
         DBX66_7 : Bool;   // 1;ROLLS T1-A;Disj. Termic Rola Nr.4 C.Role T1-A Declansat;DI;W2;1;M
         DBX67_0 : Bool;   // 1;ROLLS T1-A;Disj. Termic Rola Nr.5 C.Role T1-A Declansat;DI;W2;1;M
         DBX67_1 : Bool;   // 1;ROLLS T1-A;Disj. Termic Rola Nr.6 C.Role T1-A Declansat;DI;W2;1;M
         DBX67_2 : Bool;   // 1;ROLLS T1-A;Disj. Termic Rola Nr.7 C.Role T1-A Declansat;DI;W2;1;M
         DBX67_3 : Bool;   // 1;ROLLS T1-A;Disj. Termic Rola Nr.8 C.Role T1-A Declansat;DI;W2;1;M
         DBX67_4 : Bool;   // 1;ROLLS T1-A;TimeOut Cuplare/Decuplare Vent.Mot. C.Role T1-A;DI;W3;1;M
         DBX67_5 : Bool;   // 1;ROLLS T1-A;Disjunctor Th. AlimVent.Mot.C.Role T1A-Declansat;DI;A1;1;M
         DBX67_6 : Bool;
         DBX67_7 : Bool;   // 1;ROLLS T1-A;TimeOut Cuplare Alim.Inverter C.Role T1-A;DI;A1;1;M;O;K
         DBX68_0 : Bool;   // 1;ROLLS T1-A;Suma Disj. Termice Vent.Mot. C.Role T1-A-Declansat;DI;A1;1;M;O
         DBX68_1 : Bool;   // 1;ROLLS T1-A;Inverter Mot. C.Role T1-A - Avarie;DI;A1;1;M;O;K
         DBX68_2 : Bool;   // 1;ROLLS T1-A;Eroare Encoder C.Role T1-A;DI;A1;1;M;O;K
         DBX68_3 : Bool;   // 1;ROLLS T1-A;Role T1-A TimeOut LB Masurare Lungime ON;SQ;A1;1;M;O
         DBX68_4 : Bool;   // 1;ROLLS T1-A;Role T1-A TimeOut LB Masurare Lungime OFF;SQ;A1;1;M;O
         DBX68_5 : Bool;
         DBX68_6 : Bool;
         DBX68_7 : Bool;
         DBX69_0 : Bool;
         DBX69_1 : Bool;
         DBX69_2 : Bool;
         DBX69_3 : Bool;
         DBX69_4 : Bool;
         DBX69_5 : Bool;
         DBX69_6 : Bool;
         DBX69_7 : Bool;
         DBX70_0 : Bool;   // 1;CHAIN T1-C;TimeOut Cuplare/Decuplare Contactor Lant T1-C;DI;A1;2;M;O;K
         DBX70_1 : Bool;
         DBX70_2 : Bool;   // 1;CHAIN T1-C;TimeOut Deplasare Lant T1-C in pozitia Pas;DI;A1;2;M;O;K
         DBX70_3 : Bool;   // 1;CHAIN T1-C;Disjunctor Termic Lant T1-C - Declansat;DI;A1;2;M;K
         DBX70_4 : Bool;   // 1;CHAIN T1-C;Sectionator Alimentare Lant T1-C - Decuplat;DI;A1;2;M;K
         DBX70_5 : Bool;   // 1;STOPPER T1-C;Disjunctor Termic Opritor T1-C - Declansat;DI;A1;2;M;K
         DBX70_6 : Bool;   // 1;STOPPER T1-C;Sectionator Alimentare Opritor T1-C - Decuplat;DI;A1;2;M;K
         DBX70_7 : Bool;   // 1;STOPPER T1-C;TimeOut Cuplare Contactor Opritor T1-C;DI;A1;2;M;O;K
         DBX71_0 : Bool;
         DBX71_1 : Bool;
         DBX71_2 : Bool;
         DBX71_3 : Bool;
         DBX71_4 : Bool;
         DBX71_5 : Bool;
         DBX71_6 : Bool;
         DBX71_7 : Bool;
         DBX72_0 : Bool;
         DBX72_1 : Bool;
         DBX72_2 : Bool;
         DBX72_3 : Bool;
         DBX72_4 : Bool;
         DBX72_5 : Bool;
         DBX72_6 : Bool;
         DBX72_7 : Bool;
         DBX73_0 : Bool;
         DBX73_1 : Bool;
         DBX73_2 : Bool;
         DBX73_3 : Bool;
         DBX73_4 : Bool;
         DBX73_5 : Bool;
         DBX73_6 : Bool;
         DBX73_7 : Bool;
         DBX74_0 : Bool;   // 1;FLIPPER T1C;Lipsa Tensiune Alimentare Aruncator T1-C;DI;A1;2;M;K
         DBX74_1 : Bool;   // 1;FLIPPER T1C;TimeOut Deplasare Aruncator T1-C in pozitia Sus;DI;A1;2;M;O
         DBX74_2 : Bool;   // 1;FLIPPER T1C;TimeOut Deplasare Aruncator T1-C in pozitia Jos;DI;A1;2;M;O
         DBX74_3 : Bool;   // 1;FLIPPER T1C;Eroare Depozitare Teava pe C.Role;SQ;A1;2;O
         DBX74_4 : Bool;
         DBX74_5 : Bool;
         DBX74_6 : Bool;
         DBX74_7 : Bool;
         DBX75_0 : Bool;
         DBX75_1 : Bool;
         DBX75_2 : Bool;
         DBX75_3 : Bool;
         DBX75_4 : Bool;
         DBX75_5 : Bool;
         DBX75_6 : Bool;
         DBX75_7 : Bool;
         DBX76_0 : Bool;
         DBX76_1 : Bool;
         DBX76_2 : Bool;
         DBX76_3 : Bool;
         DBX76_4 : Bool;
         DBX76_5 : Bool;
         DBX76_6 : Bool;
         DBX76_7 : Bool;
         DBX77_0 : Bool;
         DBX77_1 : Bool;
         DBX77_2 : Bool;
         DBX77_3 : Bool;
         DBX77_4 : Bool;
         DBX77_5 : Bool;
         DBX77_6 : Bool;
         DBX77_7 : Bool;
         DBX78_0 : Bool;   // 1;ROLLS T1-C;Suma Disjuntoare Termice C.Role T1-C Declansat;DI;A1;2;M;K
         DBX78_1 : Bool;   // 1;ROLLS T1-C;Sectionator Alim.Inverter C.Role T1-C Decuplat;DI;A2;2;M;K
         DBX78_2 : Bool;   // 1;ROLLS T1-C;Lipsa Tensiune de Comanda C.Role T1-C;DI;A2;2;M;K
         DBX78_3 : Bool;   // 1;ROLLS T1-C;TimeOut Rotire Role C.Role T1-C;DI;A1;2;M;O;K
         DBX78_4 : Bool;   // 1;ROLLS T1-C;Disjunctor Termic Rola Nr.1 C.Role T1-C Declansat;DI;W2;2;M
         DBX78_5 : Bool;   // 1;ROLLS T1-C;Disjunctor Termic Rola Nr.2 C.Role T1-C Declansat;DI;W2;2;M
         DBX78_6 : Bool;   // 1;ROLLS T1-C;Disjunctor Termic Rola Nr.3 C.Role T1-C Declansat;DI;W2;2;M
         DBX78_7 : Bool;   // 1;ROLLS T1-C;Disjunctor Termic Rola Nr.4 C.Role T1-C Declansat;DI;W2;2;M
         DBX79_0 : Bool;   // 1;ROLLS T1-C;Disjunctor Termic Rola Nr.5 C.Role T1-C Declansat;DI;W2;2;M
         DBX79_1 : Bool;   // 1;ROLLS T1-C;Disjunctor Termic Rola Nr.6 C.Role T1-C Declansat;DI;W2;2;M
         DBX79_2 : Bool;   // 1;ROLLS T1-C;Disjunctor Termic Rola Nr.7 C.Role T1-C Declansat;DI;W2;2;M
         DBX79_3 : Bool;   // 1;ROLLS T1-C;Disjunctor Termic Rola Nr.8 C.Role T1-C Declansat;DI;W2;2;M
         DBX79_4 : Bool;   // 1;ROLLS T1-C;Disjunctor Termic Rola Nr.9 C.Role T1-C Declansat;DI;W2;2;M
         DBX79_5 : Bool;   // 1;ROLLS T1-C;Disjunctor Termic Rola Nr10 C.Role T1-C Declansat;DI;W2;2;M
         DBX79_6 : Bool;   // 1;ROLLS T1-C;Disjunctor Termic Rola Nr11 C.Role T1-C Declansat;DI;W2;2;M
         DBX79_7 : Bool;   // 1;ROLLS T1-C;Disjunctor Termic Rola Nr12 C.Role T1-C Declansat;DI;W2;2;M
         DBX80_0 : Bool;   // 1;ROLLS T1-C;Disjunctor Termic Rola Nr13 C.Role T1-C Declansat;DI;W2;2;M
         DBX80_1 : Bool;   // 1;ROLLS T1-C;Eroare Encoder C.Role T1-C;DI;A2;2;M;O;K
         DBX80_2 : Bool;   // 1;ROLLS T1-C;Disjunctor Termic Vent.Mot C.Role T1C Declansat;DI;A1;2;M
         DBX80_3 : Bool;   // 1;ROLLS T1-C;TimeOut Cuplare/Decuplare Vent.Mot C.Role T1-C;DI;A1;2;M;O
         DBX80_4 : Bool;   // 1;ROLLS T1-C;TimeOut Cuplare Alim.InverterC.Role T1-C;DI;A1;2;M;O;K
         DBX80_5 : Bool;   // 1;ROLLS T1-C;Inverter Mot. C.Role T1-C Avarie;DI;A1;2;M;O;K
         DBX80_6 : Bool;   // 1;ROLLS T1-C;Role T1-C TimeOut LB Masurare Lungime ON;SQ;A1;2;M;O
         DBX80_7 : Bool;   // 1;ROLLS T1-C;Role T1-C TimeOut LB Masurare Lungime OFF;SQ;A1;2;M;O
         DBX81_0 : Bool;
         DBX81_1 : Bool;
         DBX81_2 : Bool;
         DBX81_3 : Bool;
         DBX81_4 : Bool;
         DBX81_5 : Bool;
         DBX81_6 : Bool;
         DBX81_7 : Bool;
         DBX82_0 : Bool;   // 10;EXCENTRIC T10;Lipsa Tensiune de Comanda Excentric T10;DI;A1;28;M;K
         DBX82_1 : Bool;   // 10;EXCENTRIC T10;Probleme Fuzibil Excentric T10;DI;A1;28;M;K
         DBX82_2 : Bool;   // 10;EXCENTRIC T10;Disjunctor Termic Mot. Excentric T10 - Declansat;DI;A1;28;M;K
         DBX82_3 : Bool;   // 10;EXCENTRIC T10;Fuzibil Neinserat Excentric T10;DI;A1;28;M;K
         DBX82_4 : Bool;   // 10;EXCENTRIC T10;Inverter Mot. Excentric T10 - Avarie;DI;A1;28;M;O;K
         DBX82_5 : Bool;   // 10;EXCENTRIC T10;Disjunctor Frana Excentric T10 - Declansat;DI;A1;28;M;K
         DBX82_6 : Bool;   // 10;EXCENTRIC T10;Disjunctor Th.AlimVent.Mot.ExcentricT10 Declansat;DI;A1;28;M
         DBX82_7 : Bool;   // 10;EXCENTRIC T10;TimeOut Deplasare Inainte/Inapoi Excentric T10;DI;A1;28;M;O;K
         DBX83_0 : Bool;   // 10;EXCENTRIC T10;TimeOut Deplasare Excentric T10 in Pozitie;DI;A1;28;M;O;K
         DBX83_1 : Bool;   // 10;EXCENTRIC T10;Comunicatie Pierduta Encoder T10;DI;A2;28;M;O;K
         DBX83_2 : Bool;   // 10;EXCENTRIC T10;Senzor Home nedetectat sau defect;DI;A1;28;M;O;K
         DBX83_3 : Bool;   // 10;EXCENTRIC T10;TimeOut Cuplare/Decuplare Vent.Mot ExcentricT10;DI;A1;28;M;O
         DBX83_4 : Bool;   // 10;EXCENTRIC T10;Eroare Depozitare Teava pe Pat Racire T10;SQ;A1;28;O
         DBX83_5 : Bool;   // 10;EXCENTRIC T10;TimeOut Cuplare/Decuplare Frana Excentric T10;DI;A1;28;M;O;K
         DBX83_6 : Bool;
         DBX83_7 : Bool;
         DBX84_0 : Bool;   // 10;CHAIN T10;Lipsa Tensiune de Comanda Lant T10;DI;A1;28;M;K
         DBX84_1 : Bool;   // 10;CHAIN T10;Probleme Fuzibil Lant T10;DI;A1;28;M;K
         DBX84_2 : Bool;   // 10;CHAIN T10;Disjunctor Termic Mot. Lant T10 - Declansat;DI;A1;28;M;K
         DBX84_3 : Bool;   // 10;CHAIN T10;Fuzibil Neinserat Lant T10;DI;A1;28;M;K
         DBX84_4 : Bool;   // 10;CHAIN T10;Inverter Mot. Lant T10 - Avarie;DI;A1;28;M;O;K
         DBX84_5 : Bool;   // 10;CHAIN T10;Disjunctor Frana Lant T10 - Declansat;DI;A1;28;M;O;K
         DBX84_6 : Bool;   // 10;CHAIN T10;Disjunctor Termic Alim. Vent.Mot. Lant T10 - Declansat;DI;A1;28;M
         DBX84_7 : Bool;   // 10;CHAIN T10;Senzor Incetinire T10 - Avarie(blocat pe "activat");DI;A1;28;M;O;K
         DBX85_0 : Bool;   // 10;CHAIN T10;TimeOut Deplasare Lant T10;DI;A1;28;M;O;K
         DBX85_1 : Bool;   // 10;CHAIN T10;Comunicatie Pierduta Encoder Lant T10;DI;A2;28;M;O;K
         DBX85_2 : Bool;   // 10;CHAIN T10;Senzor home nedetectat sau defect;DI;A1;28;M;O;K
         DBX85_3 : Bool;   // 10;CHAIN T10;TimeOut Cuplare/Decuplare Alim.Inv. Lant T10;DI;A1;28;M;O;K
         DBX85_4 : Bool;   // 10;CHAIN T10;TimeOut Deplasare Lant T10 in pozitia Pas;DI;A1;28;M;O;K
         DBX85_5 : Bool;   // 10;CHAIN T10;Eroare Depozitare Teava pe Opritor dupa Lant T10;DI;A1;28;O
         DBX85_6 : Bool;   // 10;CHAIN T10;TimeOut Cuplare/Decuplare Frana Lant T10;DI;A1;28;M;O;K
         DBX85_7 : Bool;
         DBX86_0 : Bool;   // 10;CHAIN T10 SPIN;Lipsa Tensiune de Comanda Rostogolire T10;DI;A2;28;M;K
         DBX86_1 : Bool;   // 10;CHAIN T10 SPIN;Probleme Fuzibil Rostogolire T10;DI;A1;28;M;K
         DBX86_2 : Bool;   // 10;CHAIN T10 SPIN;Disjunctor Lant Rostogolire T10;DI;A1;28;M;K
         DBX86_3 : Bool;   // 10;CHAIN T10 SPIN;Fuzibil Neinserat Rostogolire T10;DI;A1;28;M;K
         DBX86_4 : Bool;   // 10;CHAIN T10 SPIN;Inverter Mot. LantRost. T10 - Avarie;DI;A1;28;M;O;K
         DBX86_5 : Bool;   // 10;CHAIN T10 SPIN;Disjunctor Frana Rostogolire T10-Declansat;DI;A1;28;M;O;K
         DBX86_6 : Bool;   // 10;CHAIN T10 SPIN;Disj. Th. AlimVent.Mot.Lant Rost T10 Declansa;DI;A1;28;M;O;K
         DBX86_7 : Bool;   // 10;CHAIN T10 SPIN;TimeOut Deplasare LantRost. T10;DI;A1;28;M;O;K
         DBX87_0 : Bool;   // 10;CHAIN T10 SPIN;TimeOut Cuplare/Decuplare Vent.Mot LantRost;DI;A1;28;M;O
         DBX87_1 : Bool;
         DBX87_2 : Bool;
         DBX87_3 : Bool;
         DBX87_4 : Bool;
         DBX87_5 : Bool;   // 10;STOPPER T10;TimeOut Deplasare Opritor T10 in pozitia Sus;DI;A1;28;O
         DBX87_6 : Bool;   // 10;STOPPER T10;TimeOut Deplasare Opritor T10 in pozitia Jos;DI;A1;28;O
         DBX87_7 : Bool;   // 10;STOPPER T10;Eroare Depozitare Teava pe C.Role T10-2;SQ;A1;28;O
         DBX88_0 : Bool;
         DBX88_1 : Bool;
         DBX88_2 : Bool;
         DBX88_3 : Bool;
         DBX88_4 : Bool;
         DBX88_5 : Bool;
         DBX88_6 : Bool;
         DBX88_7 : Bool;
         DBX89_0 : Bool;
         DBX89_1 : Bool;
         DBX89_2 : Bool;
         DBX89_3 : Bool;
         DBX89_4 : Bool;   // 4;ROLLS T3;Coliziune teava in Calitor;DI;A3;8;M;O
         DBX89_5 : Bool;   // 4;ROLLS T3;Disjunctor Termic Vent.Mot. C.Role T3 - Declansat;DI;A1;8;M
         DBX89_6 : Bool;   // 4;ROLLS T3;Inverter Mot. C.Role T3 - Avarie;DI;A1;8;M;O;K
         DBX89_7 : Bool;   // 4;ROLLS T3;TimeOut Cuplare/Decuplare Vent.Mot. C.Role T3;DI;A1;8;M;O
         DBX90_0 : Bool;   // 4;ROLLS T3;Lipsa Tensiune de Comanda C.Role T3;DI;A1;8;M;K
         DBX90_1 : Bool;   // 4;ROLLS T3;Sectionator Alim.Inverter Mot. C.Role T3-Decuplat;DI;A1;8;M;K
         DBX90_2 : Bool;   // 4;ROLLS T3;Suma Disjunctoare Termice Mot.C.Role T3-Declansat;DI;A1;8;M;K
         DBX90_3 : Bool;   // 4;ROLLS T3;Disjunctor Termic Rola Nr.1 C.Role T3 Declansat;DI;W2;8;M
         DBX90_4 : Bool;   // 4;ROLLS T3;Disjunctor Termic Rola Nr.2 C.Role T3 Declansat;DI;W2;8;M
         DBX90_5 : Bool;   // 4;ROLLS T3;Disjunctor Termic Rola Nr.3 C.Role T3 Declansat;DI;W2;8;M
         DBX90_6 : Bool;   // 4;ROLLS T3;Disjunctor Termic Rola Nr.4 C.Role T3 Declansat;DI;W2;8;M
         DBX90_7 : Bool;   // 4;ROLLS T3;Disjunctor Termic Rola Nr.5 C.Role T3 Declansat;DI;W2;8;M
         DBX91_0 : Bool;   // 4;ROLLS T3;TimeOut Rotire Role C.Role T3;DI;A1;8;M;O;K
         DBX91_1 : Bool;   // 4;ROLLS T3;TimeOut Cuplare/Decuplare Alim.Inv. C.Role T3;DI;A1;8;M;O;K
         DBX91_2 : Bool;   // 4;DEZTUNDERIZATOR;Disjunctor Term. Deztunderizator-Declansat;DI;A2;7;M;O;K
         DBX91_3 : Bool;   // 4;DEZTUNDERIZATOR;Sectionator Alim. Deztunderizator-Decuplat;DI;A1;7;M;K
         DBX91_4 : Bool;   // 4;DEZTUNDERIZATOR;SoftStarter SIKO Destunderizator - Avarie;DI;A2;7;M;O;K
         DBX91_5 : Bool;
         DBX91_6 : Bool;   // 4;DEZTUNDERIZATOR;Lipsa Tensiune de Comanda Deztunderizator;DI;A1;7;M;O;K
         DBX91_7 : Bool;   // 4;HEADHARD1;Disjunctor Termic Mot. Cap Calire Nr.1-Declansat;DI;A1;8;M;K
         DBX92_0 : Bool;   // 4;HEADHARD1;Disj. Termic Alim. Mot. Cap Calire Nr.1-Decuplat;DI;A1;8;M;K
         DBX92_1 : Bool;   // 4;HEADHARD1;TimeOut Deplasare Cap Calire Nr.1;DI;A1;8;M;O
         DBX92_2 : Bool;   // 4;DEZTUNDERIZATOR;Lipsa Tensiune Alimentare 24V Deztunder;DI;A1;8;M;K
         DBX92_3 : Bool;   // 4;HEADHARD2;Disjunctor Termic Mot. Cap Calire Nr.2-Declansat;DI;A1;8;M;K
         DBX92_4 : Bool;   // 4;HEADHARD2;Disj. Termic Alim. Mot. Cap Calire Nr.2-Decuplat;DI;A1;8;M;K
         DBX92_5 : Bool;   // 4;HEADHARD2;TimeOut Deplasare Cap Calire Nr.2;DI;A1;8;M;O
         DBX92_6 : Bool;
         DBX92_7 : Bool;   // 4;HEADHARD3;Disjunctor Termic Mot. Cap Calire Nr.3-Declansat;DI;A1;8;M;K
         DBX93_0 : Bool;   // 4;HEADHARD3;Disj. Termic Alim. Mot. Cap Calire Nr.3-Decuplat;DI;A1;8;M;K
         DBX93_1 : Bool;   // 4;HEADHARD3;TimeOut Deplasare Cap Calire Nr.3;DI;A1;8;M;O
         DBX93_2 : Bool;
         DBX93_3 : Bool;   // 4;BEAM;Disjunctor Termic Mot. Grinda - Declansat;DI;A1;8;M;K
         DBX93_4 : Bool;   // 4;BEAM;Disjunctor Termic Alim. Mot. Grinda - Decuplat;DI;A1;8;M;K
         DBX93_5 : Bool;   // 4;BEAM;BEAN:TimeOut Deplasare Grinda;DI;A1;8;M;O
         DBX93_6 : Bool;   // 4;BEAM;Lipsa Tensiune Comanda Grinda/Deztunderizator;DI;A1;8;M;K
         DBX93_7 : Bool;   // 4;ROLLS T3;Suma Disj. Termice Vent.Mot. C.Role T3 - Declansat;DI;A1;8;M
         DBX94_0 : Bool;   // 4;ROLLS T4-1;Suma Disj. Termice Mot. C.Role T4-1 - Declansat;DI;A1;10;M;K
         DBX94_1 : Bool;   // 4;ROLLS T4-1;Sectionator Alim.Inv. Mot. C.Role T4-1-Decuplat;DI;A1;10;M;K
         DBX94_2 : Bool;   // 4;ROLLS T4-1;Lipsa Tensiune de Comanda C.Role T4-1;DI;A1;10;M;K
         DBX94_3 : Bool;   // 4;ROLLS T4-1;TimeOut Rotire Role C.Role T4-1;DI;A1;10;M;O;K
         DBX94_4 : Bool;   // 4;ROLLS T4-1;Disj. Termic Rola Nr.1 C.Role T4-1 Declansat;DI;W2;10;M
         DBX94_5 : Bool;   // 4;ROLLS T4-1;Disj. Termic Rola Nr.2 C.Role T4-1 Declansat;DI;W2;10;M
         DBX94_6 : Bool;   // 4;ROLLS T4-1;Disj. Termic Rola Nr.3 C.Role T4-1 Declansat;DI;W2;10;M
         DBX94_7 : Bool;   // 4;ROLLS T4-1;Disj. Termic Rola Nr.4 C.Role T4-1 Declansat;DI;W2;10;M
         DBX95_0 : Bool;   // 4;ROLLS T4-1;Disj. Termic Rola Nr.5 C.Role T4-1 Declansat;DI;W2;10;M
         DBX95_1 : Bool;   // 4;ROLLS T4-1;Disj. Termic Rola Nr.6 C.Role T4-1 Declansat;DI;W2;10;M
         DBX95_2 : Bool;   // 4;ROLLS T4-1;Disj. Termic Rola Nr.7 C.Role T4-1 Declansat;DI;W2;10;M
         DBX95_3 : Bool;   // 4;ROLLS T4-1;Disj. Termic Rola Nr.8 C.Role T4-1 Declansat;DI;W2;10;M
         DBX95_4 : Bool;   // 4;ROLLS T4-1;Disj. Termic Rola Nr.9 C.Role T4-1 Declansat;DI;W2;10;M
         DBX95_5 : Bool;   // 4;ROLLS T4-1;Disjunctor Th. AlimVent.Mot.C.Role T4-1 Declansat;DI;A1;10;M
         DBX95_6 : Bool;   // 4;ROLLS T4-1;Role T4-1 TimeOut Pozitionare Teava;SQ;A1;10;O
         DBX95_7 : Bool;
         DBX96_0 : Bool;
         DBX96_1 : Bool;
         DBX96_2 : Bool;   // 4;ROLLS T4-1;Suma Disj. Th. Vent.Mot. C.Role T4-1-Declansat;DI;A1;10;M
         DBX96_3 : Bool;   // 4;ROLLS T4-1;TimeOut Cuplare/Decuplare Vent.Mot.C.Role T4-1;DI;A1;10;M;O
         DBX96_4 : Bool;   // 4;ROLLS T4-1;TimeOut Cuplare Alim.Inv. C.Role T4-1;DI;A1;10;M;O;K
         DBX96_5 : Bool;   // 4;ROLLS T4-1;Inverter Mot. C.Role T4-1 - Avarie;DI;A1;10;M;O;K
         DBX96_6 : Bool;
         DBX96_7 : Bool;
         DBX97_0 : Bool;   // 4;DEZTUNDERIZATOR;Disjunctor Termic Pompa 9.1 - Declansat;DI;A1;7;M;K
         DBX97_1 : Bool;   // 4;DEZTUNDERIZATOR;Disjunctor Termic Pompa 9.2 - Declansat;DI;A1;7;M;K
         DBX97_2 : Bool;   // 4;DEZTUNDERIZATOR;Lipsa confirm. cuplare contactor Pompa 9.1;DI;A1;7;M;K
         DBX97_3 : Bool;   // 4;DEZTUNDERIZATOR;Lipsa confirm. cuplare contactor Pompa 9.2;DI;A1;7;M;K
         DBX97_4 : Bool;   // 4;DEZTUNDERIZATOR;Sistem Oprire de Urgenta Hammelman-Declansat;EM;A1;7;M;O;K
         DBX97_5 : Bool;   // 4;DEZTUNDERIZATOR;Alarma generala Unitate Hammelmann;DI;A1;7;M;O;K
         DBX97_6 : Bool;   // 4;DEZTUNDERIZATOR;Lipsa confirm robinet izolare deschis 100bar;DI;A1;7;M;O;K
         DBX97_7 : Bool;   // 4;DEZTUNDERIZATOR;Lipsa confirm robinet izolare deschis 180bar;DI;A1;7;M;O;K
         DBX98_0 : Bool;   // 4;EXCENTRIC T4;TimeOut Deplasare Inainte Excentric T4;DI;A1;10;M;O;K
         DBX98_1 : Bool;   // 4;EXCENTRIC T4;TimeOut Deplasare Inapoi Excentric T4;DI;A1;10;M;O;K
         DBX98_2 : Bool;   // 4;EXCENTRIC T4;TimeOut Deplasare Excentric T4 in Pozitie;DI;A1;10;M;O;K
         DBX98_3 : Bool;   // 4;EXCENTRIC T4;Disjunctor Termic Mot. Excentric T4-Declansat;DI;A1;10;M;K
         DBX98_4 : Bool;   // 4;EXCENTRIC T4;Alim. SoftStarter SIKO Excentric T4-Decuplat;DI;A1;10;M;K
         DBX98_5 : Bool;   // 4;EXCENTRIC T4;Alim. Frana Mot. Excentric T4 - Decuplat;DI;A1;10;M;K
         DBX98_6 : Bool;   // 4;EXCENTRIC T4;Lipsa Tensiune de Comanda Excentric T4;DI;A1;10;M;K
         DBX98_7 : Bool;   // 4;EXCENTRIC T4;SoftStarter SIKO Excentric T4 - Avarie;DI;A1;10;M;O;K
         DBX99_0 : Bool;   // 4;EXCENTRIC T4;Eroare Depozitare Teava pe Pat Racire T4;SQ;A1;10;O
         DBX99_1 : Bool;
         DBX99_2 : Bool;
         DBX99_3 : Bool;
         DBX99_4 : Bool;
         DBX99_5 : Bool;
         DBX99_6 : Bool;
         DBX99_7 : Bool;
         DBX100_0 : Bool;   // 4;DEZTUNDERIZATOR;Presiune prea mica inainte de P. Hammelmann;DI;A1;7;O;K
         DBX100_1 : Bool;   // 4;DEZTUNDERIZATOR;Presiune prea mare dupa unit joasa pres.;DI;A1;7;O;K
         DBX100_2 : Bool;   // 4;DEZTUNDERIZATOR;Lipsa confirmare curgere pe alimentare;DI;A1;7;M;O;K
         DBX100_3 : Bool;
         DBX100_4 : Bool;
         DBX100_5 : Bool;
         DBX100_6 : Bool;
         DBX100_7 : Bool;
         DBX101_0 : Bool;
         DBX101_1 : Bool;
         DBX101_2 : Bool;
         DBX101_3 : Bool;
         DBX101_4 : Bool;
         DBX101_5 : Bool;
         DBX101_6 : Bool;
         DBX101_7 : Bool;
         DBX102_0 : Bool;   // 4;CHAIN T4;Stop Permisie Cuplare Lant T4 - Actionat;DI;A1;10;M;O;K
         DBX102_1 : Bool;   // 4;CHAIN T4;TimeOut Cuplare/Decuplare Alim.Inv. Lant T4;DI;A1;10;M;O;K
         DBX102_2 : Bool;   // 4;CHAIN T4;Lipsa Tensiune de Comanda Lant T4;DI;A1;10;M;K
         DBX102_3 : Bool;   // 4;CHAIN T4;Sectionator Alim.Inv. Mot. Lant T4 - Decuplat;DI;A1;10;M;K
         DBX102_4 : Bool;   // 4;CHAIN T4;Alim. Frana Mot. Lant T4 - Decuplat;DI;A1;10;M;K
         DBX102_5 : Bool;   // 4;CHAIN T4;Inverter Mot. Lant T4 - Avarie;DI;A1;10;M;O;K
         DBX102_6 : Bool;   // 4;CHAIN T4 SPIN;TimeOut Cuplare/Decupl. Alim.Inv.LantRost. T4;DI;A1;10;M;O;K
         DBX102_7 : Bool;   // 4;CHAIN T4 SPIN;Sectionator Alim.Inv Mot.LantRost T4-Decuplat;DI;A1;10;M;K
         DBX103_0 : Bool;   // 4;CHAIN T4 SPIN;Disjunctor Termic Mot. LantRost. T4-Declansat;DI;A1;10;M;K
         DBX103_1 : Bool;   // 4;CHAIN T4;TimeOut Deplasare Lant T4 in pozitia Pas;DI;A1;10;M;O;K
         DBX103_2 : Bool;   // 4;CHAIN T4 SPIN;Inverter Mot. LantRost. T4 - Avarie;DI;A1;10;M;O;K
         DBX103_3 : Bool;   // 4;CHAIN T4 SPIN;Stop Permisie Cuplare LantRost. T4 - Actionat;DI;A1;10;M;O;K
         DBX103_4 : Bool;   // 4;CHAIN T4;TimeOut Deplasare Lant T4;DI;A1;10;M;O;K
         DBX103_5 : Bool;   // 4;CHAIN T4;TimeOut Cuplare/Decuplare Frana Lant T4;DI;A1;10;M;O;K
         DBX103_6 : Bool;   // 4;CHAIN T4 SPIN;TimeOut Deplasare LantRost. T4;DI;A1;10;M;O;K
         DBX103_7 : Bool;   // 4;CHAIN T4;Disjunctor Termic Alim. Vent.Mot. Lant T4-Declansat;DI;A1;10;M
         DBX104_0 : Bool;
         DBX104_1 : Bool;
         DBX104_2 : Bool;
         DBX104_3 : Bool;   // 4;CHAIN T4;Eroare Depozitare Teava pe Opritor dupa Lant T4;DI;A1;10;O
         DBX104_4 : Bool;   // 4;CHAIN T4;Senzor Incetinire T4 - Avarie(blocat pe "activat");DI;A1;10;M;O;K
         DBX104_5 : Bool;
         DBX104_6 : Bool;
         DBX104_7 : Bool;
         DBX105_0 : Bool;
         DBX105_1 : Bool;
         DBX105_2 : Bool;
         DBX105_3 : Bool;
         DBX105_4 : Bool;
         DBX105_5 : Bool;
         DBX105_6 : Bool;
         DBX105_7 : Bool;
         DBX106_0 : Bool;   // 4;STOPPER T4;Lipsa Tensiune Alimentare Opritor T4;DI;A1;10;M;K
         DBX106_1 : Bool;   // 4;STOPPER T4;TimeOut Deplasare Opritor T4 in pozitia Sus;DI;A1;10;O
         DBX106_2 : Bool;   // 4;STOPPER T4;TimeOut Deplasare Opritor T4 in pozitia Jos;DI;A1;10;O
         DBX106_3 : Bool;   // 4;STOPPER T4;Eroare Depozitare Teava pe C.Role T4-1;SQ;A1;10;O
         DBX106_4 : Bool;
         DBX106_5 : Bool;
         DBX106_6 : Bool;
         DBX106_7 : Bool;
         DBX107_0 : Bool;
         DBX107_1 : Bool;
         DBX107_2 : Bool;
         DBX107_3 : Bool;
         DBX107_4 : Bool;
         DBX107_5 : Bool;
         DBX107_6 : Bool;
         DBX107_7 : Bool;
         DBX108_0 : Bool;
         DBX108_1 : Bool;
         DBX108_2 : Bool;
         DBX108_3 : Bool;
         DBX108_4 : Bool;
         DBX108_5 : Bool;
         DBX108_6 : Bool;
         DBX108_7 : Bool;
         DBX109_0 : Bool;
         DBX109_1 : Bool;
         DBX109_2 : Bool;
         DBX109_3 : Bool;
         DBX109_4 : Bool;
         DBX109_5 : Bool;
         DBX109_6 : Bool;
         DBX109_7 : Bool;
         DBX110_0 : Bool;   // 4;ROLLS T4-2;Suma Disj. Termice Mot. C.Role T4-2 Declansat;DI;A1;10;M;K
         DBX110_1 : Bool;   // 4;ROLLS T4-2;Sectionator Alim.Inv. Mot. C.Role T4-2 Decuplat;DI;A1;10;M;K
         DBX110_2 : Bool;   // 4;ROLLS T4-2;Lipsa Tensiune de Comanda C.Role T4-2;DI;A1;10;M;K
         DBX110_3 : Bool;   // 4;ROLLS T4-2;Timeout Rotire Role C.Role T4-2;DI;A1;10;M;O;K
         DBX110_4 : Bool;   // 4;ROLLS T4-2;Disj. Termic Rola Nr.1 C.Role T4-2 Declansat;DI;W2;10;M
         DBX110_5 : Bool;   // 4;ROLLS T4-2;Disj. Termic Rola Nr.2 C.Role T4-2 Declansat;DI;W2;10;M
         DBX110_6 : Bool;   // 4;ROLLS T4-2;Disj. Termic Rola Nr.3 C.Role T4-2 Declansat;DI;W2;10;M
         DBX110_7 : Bool;   // 4;ROLLS T4-2;Disj. Termic Rola Nr.4 C.Role T4-2 Declansat;DI;W2;10;M
         DBX111_0 : Bool;   // 4;ROLLS T4-2;Disj. Termic Rola Nr.5 C.Role T4-2 Declansat;DI;W2;10;M
         DBX111_1 : Bool;   // 4;ROLLS T4-2;Disj. Termic Rola Nr.6 C.Role T4-2 Declansat;DI;W2;10;M
         DBX111_2 : Bool;   // 4;ROLLS T4-2;Disj. Termic Rola Nr.7 C.Role T4-2 Declansat;DI;W2;10;M
         DBX111_3 : Bool;   // 4;ROLLS T4-2;Disj. Termic Rola Nr.8 C.Role T4-2 Declansat;DI;W2;10;M
         DBX111_4 : Bool;   // 4;ROLLS T4-2;Disj. Termic Rola Nr.9 C.Role T4-2 Declansat;DI;W2;10;M
         DBX111_5 : Bool;   // 4;ROLLS T4-2;Inverter Mot. C.Role T4-2 Avarie;DI;A1;10;M;O;K
         DBX111_6 : Bool;   // 4;ROLLS T4-2;Disjunctor Th. AlimVent.Mot.C.Role T4-2 Declansat;DI;A1;10;M
         DBX111_7 : Bool;   // 4;ROLLS T4-2;Role T4-2 TimeOut Prezenta Teava ON;SQ;A1;10;O
         DBX112_0 : Bool;   // 4;ROLLS T4-2;Role T4-2 TimeOut Prezenta Teava OFF;SQ;A1;10;O
         DBX112_1 : Bool;
         DBX112_2 : Bool;   // 4;ROLLS T4-2;Suma Disj. Th. Vent.Mot. C.Role T4-2-Declansat;DI;A1;10;M
         DBX112_3 : Bool;   // 4;ROLLS T4-2;TimeOut Cuplare/Decuplare Vent.Mot. C.Role T4-2;DI;A1;10;M;O
         DBX112_4 : Bool;   // 4;ROLLS T4-2;TimeOut Cuplare/Decuplare Alim.Inv. C.Role T4-2;DI;A1;10;M;O;K
         DBX112_5 : Bool;
         DBX112_6 : Bool;
         DBX112_7 : Bool;
         DBX113_0 : Bool;
         DBX113_1 : Bool;
         DBX113_2 : Bool;
         DBX113_3 : Bool;
         DBX113_4 : Bool;
         DBX113_5 : Bool;
         DBX113_6 : Bool;
         DBX113_7 : Bool;
         DBX114_0 : Bool;   // 4;FLIPPER T1-E;Lipsa Tensiune Alimentare Aruncator T1-E;DI;A1;12;M;K
         DBX114_1 : Bool;   // 4;FLIPPER T1-E;TimeOut Deplasare Aruncator T1-E pozitia Sus;DI;A1;12;M;O
         DBX114_2 : Bool;   // 4;FLIPPER T1-E;TimeOut Deplasare Aruncator T1-E pozitia Jos;DI;A1;12;M;O
         DBX114_3 : Bool;   // 4;STOPPER T1-E;Disjunctor Termic Opritor T1-E - Declansat;DI;A1;12;M;K
         DBX114_4 : Bool;   // 4;STOPPER T1-E;Sectionator Alimentare Opritor T1-E-Decuplat;DI;A1;12;M;K
         DBX114_5 : Bool;   // 4;STOPPER T1-E;TimeOut Cuplare Contactor Opritor T1-E;DI;A1;12;M;O;K
         DBX114_6 : Bool;   // 4;STOPPER T1-E;Lipsa Tensiune de Comanda Opritor T1-E;DI;A1;12;M;K
         DBX114_7 : Bool;   // 4;FLIPPER T1-E;Disjunctor Termic Dozator T1-E - Declansat;DI;A1;12;M;K
         DBX115_0 : Bool;
         DBX115_1 : Bool;
         DBX115_2 : Bool;
         DBX115_3 : Bool;
         DBX115_4 : Bool;
         DBX115_5 : Bool;
         DBX115_6 : Bool;
         DBX115_7 : Bool;
         DBX116_0 : Bool;   // 10;ROLLS T10-2;Lipsa Tensiune de Comanda C.Role T10-2;DI;A1;28;M;K
         DBX116_1 : Bool;   // 10;ROLLS T10-2;Probleme Fuzibil C.Role T10-2;DI;A1;28;M;K
         DBX116_2 : Bool;   // 10;ROLLS T10-2;Disj. Termic Mot. C.Role T10-2 Declansat;DI;A1;28;M;K
         DBX116_3 : Bool;   // 10;ROLLS T10-2;Fuzibil Neinserat C.Role T10-2;DI;A1;28;M;K
         DBX116_4 : Bool;   // 10;ROLLS T10-2;Inverter Mot. C.Role T10-2 Avarie;DI;A1;28;M;O;K
         DBX116_5 : Bool;   // 10;ROLLS T10-2;Role T10-2 TimeOut Prezenta Teava ON;SQ;A1;28;O
         DBX116_6 : Bool;   // 10;ROLLS T10-2;Role T10-2 TimeOut Prezenta Teava OFF;SQ;A1;28;O
         DBX116_7 : Bool;   // 10;ROLLS T10-2;Timeout Rotire Role C.Role T10-2;DI;A1;28;M;O;K
         DBX117_0 : Bool;   // 10;ROLLS T10-2;TimeOut Cuplare/Decuplare Vent.Mot. C.Role T10-2;DI;A1;28;M;O
         DBX117_1 : Bool;   // 10;ROLLS T10-2;Disjunctor Th. AlimVent.Mot.C.Role T10-2 Declansat;DI;A1;28;M
         DBX117_2 : Bool;
         DBX117_3 : Bool;
         DBX117_4 : Bool;
         DBX117_5 : Bool;
         DBX117_6 : Bool;
         DBX117_7 : Bool;
         DBX118_0 : Bool;   // 4;TAMPON KASTO Cabina;Tampon Blocat la Introducere in Linie;DI;A1;11;M;O
         DBX118_1 : Bool;   // 4;TAMPON KASTO Cabina;Tampon Blocat la Scoatere in Linie;DI;A1;11;M;O
         DBX118_2 : Bool;
         DBX118_3 : Bool;
         DBX118_4 : Bool;   // 5;TAMPON KASTO T6;Tampon Blocat la Introducere in Linie;DI;A1;15;M;O
         DBX118_5 : Bool;   // 5;TAMPON KASTO T6;Tampon Blocat la Scoatere in Linie;DI;A1;15;M;O
         DBX118_6 : Bool;
         DBX118_7 : Bool;
         DBX119_0 : Bool;
         DBX119_1 : Bool;
         DBX119_2 : Bool;
         DBX119_3 : Bool;
         DBX119_4 : Bool;
         DBX119_5 : Bool;
         DBX119_6 : Bool;
         DBX119_7 : Bool;
         DBX120_0 : Bool;
         DBX120_1 : Bool;
         DBX120_2 : Bool;
         DBX120_3 : Bool;
         DBX120_4 : Bool;
         DBX120_5 : Bool;
         DBX120_6 : Bool;
         DBX120_7 : Bool;
         DBX121_0 : Bool;
         DBX121_1 : Bool;
         DBX121_2 : Bool;
         DBX121_3 : Bool;
         DBX121_4 : Bool;
         DBX121_5 : Bool;
         DBX121_6 : Bool;
         DBX121_7 : Bool;
         DBX122_0 : Bool;   // 4;ROLLS T5-1;Suma Disj. Termice Mot. C.Role T5-1 - Declansat;DI;A1;14;M;K
         DBX122_1 : Bool;   // 4;ROLLS T5-1;Sectionator Alim.Inv. Mot. C.Role T5-1-Decuplat;DI;A1;14;M;K
         DBX122_2 : Bool;   // 4;ROLLS T5-1;Lipsa Tensiune de Comanda C.Role T5-1;DI;A1;14;M;K
         DBX122_3 : Bool;   // 4;ROLLS T5-1;TimeOut Rotire Role C.Role T5-1;DI;A1;14;M;O;K
         DBX122_4 : Bool;   // 4;ROLLS T5-1;Disj. Termic Rola Nr.1 C.Role T5-1 Declansat;DI;W2;14;M
         DBX122_5 : Bool;   // 4;ROLLS T5-1;Disj. Termic Rola Nr.2 C.Role T5-1 Declansat;DI;W2;14;M
         DBX122_6 : Bool;   // 4;ROLLS T5-1;Disj. Termic Rola Nr.3 C.Role T5-1 Declansat;DI;W2;14;M
         DBX122_7 : Bool;   // 4;ROLLS T5-1;Disj. Termic Rola Nr.4 C.Role T5-1 Declansat;DI;W2;14;M
         DBX123_0 : Bool;   // 4;ROLLS T5-1;Disj. Termic Rola Nr.5 C.Role T5-1 Declansat;DI;W2;14;M
         DBX123_1 : Bool;   // 4;ROLLS T5-1;Disj. Termic Rola Nr.6 C.Role T5-1 Declansat;DI;W2;14;M
         DBX123_2 : Bool;   // 4;ROLLS T5-1;Disj. Termic Rola Nr.7 C.Role T5-1 Declansat;DI;W2;14;M
         DBX123_3 : Bool;   // 4;ROLLS T5-1;Disj. Termic Rola Nr.8 C.Role T5-1 Declansat;DI;W2;14;M
         DBX123_4 : Bool;
         DBX123_5 : Bool;   // 4;ROLLS T5-1;Suma Disj. Th. Vent.Mot. C.Role T5-1 - Declansat;DI;A1;14;M
         DBX123_6 : Bool;   // 4;ROLLS T5-1;Role T5-1 TimeOut Prezenta Teava;SQ;A1;14;O
         DBX123_7 : Bool;   // 4;ROLLS T5-1;Role T5-1 TimeOut Pozitionare Teava;SQ;A1;14;O
         DBX124_0 : Bool;
         DBX124_1 : Bool;
         DBX124_2 : Bool;   // 4;ROLLS T5-1;Disj. Th. Alim.Vent.Mot. C.Role T5-1-Declansat;DI;A1;14;M
         DBX124_3 : Bool;   // 4;ROLLS T5-1;TimeOut Cuplare/Decuplare Vent.Mot. C.Role T5-1;DI;A1;14;M;O
         DBX124_4 : Bool;   // 4;ROLLS T5-1;TimeOut Cuplare/Decuplare Alim.Inv. C.Role T5-1;DI;A1;14;M;O;K
         DBX124_5 : Bool;   // 4;ROLLS T5-1;Inverter Mot. C.Role T5-1 - Avarie;DI;A1;14;M;O;K
         DBX124_6 : Bool;
         DBX124_7 : Bool;
         DBX125_0 : Bool;
         DBX125_1 : Bool;
         DBX125_2 : Bool;
         DBX125_3 : Bool;
         DBX125_4 : Bool;
         DBX125_5 : Bool;
         DBX125_6 : Bool;
         DBX125_7 : Bool;
         DBX126_0 : Bool;   // 4;EXCENTRIC T5;TimeOut Deplasare Inainte Excentric T5;DI;A1;14;M;O;K
         DBX126_1 : Bool;   // 4;EXCENTRIC T5;TimeOut Deplasare Inapoi Excentric T5;DI;A1;14;M;O;K
         DBX126_2 : Bool;   // 4;EXCENTRIC T5;TimeOut Deplasare Excentric T5 in Pozitie;DI;A1;14;M;O;K
         DBX126_3 : Bool;   // 4;EXCENTRIC T5;Disjunctor Termic Mot. Excentric T5-Declansat;DI;A1;14;M;K
         DBX126_4 : Bool;   // 4;EXCENTRIC T5;Alim. SoftStarter SIKO Excentric T5-Decuplat;DI;A1;14;M;K
         DBX126_5 : Bool;   // 4;EXCENTRIC T5;Alim. Frana Mot. Excentric T5 - Decuplat;DI;A1;14;M;K
         DBX126_6 : Bool;   // 4;EXCENTRIC T5;Lipsa Tensiune de Comanda Excentric T5;DI;A1;14;M;K
         DBX126_7 : Bool;   // 4;EXCENTRIC T5;SoftStarter SIKO Excentric T5 - Avarie;DI;A1;14;M;O;K
         DBX127_0 : Bool;   // 4;EXCENTRIC T5;Eroare Depozitare Teava pe Pat Racire T5;SQ;A1;14;O
         DBX127_1 : Bool;
         DBX127_2 : Bool;
         DBX127_3 : Bool;
         DBX127_4 : Bool;
         DBX127_5 : Bool;
         DBX127_6 : Bool;
         DBX127_7 : Bool;
         DBX128_0 : Bool;
         DBX128_1 : Bool;
         DBX128_2 : Bool;
         DBX128_3 : Bool;
         DBX128_4 : Bool;
         DBX128_5 : Bool;
         DBX128_6 : Bool;
         DBX128_7 : Bool;
         DBX129_0 : Bool;
         DBX129_1 : Bool;
         DBX129_2 : Bool;
         DBX129_3 : Bool;
         DBX129_4 : Bool;
         DBX129_5 : Bool;
         DBX129_6 : Bool;
         DBX129_7 : Bool;
         DBX130_0 : Bool;   // 4;CHAIN T5;TimeOut Cuplare/Decuplare Alim.Inv. Lant T5;DI;A1;14;M;O;K
         DBX130_1 : Bool;   // 4;CHAIN T5;Disjunctor Termic Alim. Vent.Mot. Lant T5-Declansat;DI;A1;14;M
         DBX130_2 : Bool;   // 4;CHAIN T5;TimeOut Deplasare Lant T5 in pozitia Pas;DI;A1;14;M;O;K
         DBX130_3 : Bool;   // 4;CHAIN T5;TimeOut Cuplare/Decuplare Frana Lant T5;DI;A1;14;M;O;K
         DBX130_4 : Bool;   // 4;CHAIN T5;Sectionator Alim.Inv. Mot. Lant T5 - Decuplat;DI;A1;14;M;K
         DBX130_5 : Bool;   // 4;CHAIN T5;Lipsa Tensiune de Comanda Lant T5;DI;A1;14;M;K
         DBX130_6 : Bool;   // 4;CHAIN T5;Inverter Mot. Lant T5 - Avarie;DI;A1;14;M;O;K
         DBX130_7 : Bool;   // 4;CHAIN T5;Stop Permisie Cuplare Lant T5 - Actionat;DI;A1;14;M;K
         DBX131_0 : Bool;   // 4;CHAIN T5;TimeOut Deplasare Lant T5;DI;A1;14;M;O;K
         DBX131_1 : Bool;
         DBX131_2 : Bool;
         DBX131_3 : Bool;   // 4;CHAIN T5;Eroare Depozitare Teava pe Opritor dupa Lant T5;DI;A1;14;O
         DBX131_4 : Bool;   // 4;CHAIN T5;Senzor Incetinire T5 - Avarie (blocat pe "activat");DI;A1;14;M;O;K
         DBX131_5 : Bool;
         DBX131_6 : Bool;
         DBX131_7 : Bool;
         DBX132_0 : Bool;
         DBX132_1 : Bool;
         DBX132_2 : Bool;
         DBX132_3 : Bool;
         DBX132_4 : Bool;
         DBX132_5 : Bool;
         DBX132_6 : Bool;
         DBX132_7 : Bool;
         DBX133_0 : Bool;
         DBX133_1 : Bool;
         DBX133_2 : Bool;
         DBX133_3 : Bool;
         DBX133_4 : Bool;
         DBX133_5 : Bool;
         DBX133_6 : Bool;
         DBX133_7 : Bool;
         DBX134_0 : Bool;   // 4;STOPPER T5;Lipsa Tensiune Alimentare Opritor T5;DI;A1;14;M;K
         DBX134_1 : Bool;   // 4;STOPPER T5;TimeOut Deplasare Opritor T5 in pozitia Sus;DI;A1;14;M;O
         DBX134_2 : Bool;   // 4;STOPPER T5;TimeOut Deplasare Opritor T5 in pozitia Jos;DI;W2;14;M;O
         DBX134_3 : Bool;   // 4;STOPPER T5;Eroare Depozitare Teava pe C.Role T5;SQ;A1;14;O
         DBX134_4 : Bool;
         DBX134_5 : Bool;
         DBX134_6 : Bool;
         DBX134_7 : Bool;
         DBX135_0 : Bool;
         DBX135_1 : Bool;
         DBX135_2 : Bool;
         DBX135_3 : Bool;
         DBX135_4 : Bool;
         DBX135_5 : Bool;
         DBX135_6 : Bool;
         DBX135_7 : Bool;
         DBX136_0 : Bool;
         DBX136_1 : Bool;
         DBX136_2 : Bool;
         DBX136_3 : Bool;
         DBX136_4 : Bool;
         DBX136_5 : Bool;
         DBX136_6 : Bool;
         DBX136_7 : Bool;
         DBX137_0 : Bool;
         DBX137_1 : Bool;
         DBX137_2 : Bool;
         DBX137_3 : Bool;
         DBX137_4 : Bool;
         DBX137_5 : Bool;
         DBX137_6 : Bool;
         DBX137_7 : Bool;
         DBX138_0 : Bool;   // 4;ROLLS T5-2;Suma Disj. Termice Mot. C.Role T5-2 - Declansat;DI;A1;14;M;K
         DBX138_1 : Bool;   // 4;ROLLS T5-2;Sectionator Alim.Inv. Mot. C.Role T5-2-Decuplat;DI;A1;14;M;K
         DBX138_2 : Bool;   // 4;ROLLS T5-2;Lipsa Tensiune de Comanda C.Role T5-2;DI;A1;14;M;K
         DBX138_3 : Bool;   // 4;ROLLS T5-2;TimeOut Rotire Role C.Role T5-2;DI;A1;14;M;O;K
         DBX138_4 : Bool;   // 4;ROLLS T5-2;Disj. Termic Rola Nr.1 C.Role T5-2 Declansat;DI;W2;14;M
         DBX138_5 : Bool;   // 4;ROLLS T5-2;Disj. Termic Rola Nr.2 C.Role T5-2 Declansat;DI;W2;14;M
         DBX138_6 : Bool;   // 4;ROLLS T5-2;Disj. Termic Rola Nr.3 C.Role T5-2 Declansat;DI;W2;14;M
         DBX138_7 : Bool;   // 4;ROLLS T5-2;Disj. Termic Rola Nr.4 C.Role T5-2 Declansat;DI;W2;14;M
         DBX139_0 : Bool;   // 4;ROLLS T5-2;Disj. Termic Rola Nr.5 C.Role T5-2 Declansat;DI;W2;14;M
         DBX139_1 : Bool;   // 4;ROLLS T5-2;Disj. Termic Rola Nr.6 C.Role T5-2 Declansat;DI;W2;14;M
         DBX139_2 : Bool;   // 4;ROLLS T5-2;Disj. Termic Rola Nr.7 C.Role T5-2 Declansat;DI;W2;14;M
         DBX139_3 : Bool;   // 4;ROLLS T5-2;Disj. Termic Rola Nr.8 C.Role T5-2 Declansat;DI;W2;14;M
         DBX139_4 : Bool;   // 4;ROLLS T5-2;Disj. Termic Rola Nr.9 C.Role T5-2 Declansat;DI;W2;14;M
         DBX139_5 : Bool;   // 4;ROLLS T5-2;Disj. Termic Rola Nr.10 C.Role T5-2 Declansat;DI;W2;14;M
         DBX139_6 : Bool;   // 4;ROLLS T5-2;Disj. Th. Alim.Vent.Mot. C.Role T5-2 - Declansat;DI;A1;14;M
         DBX139_7 : Bool;   // 4;ROLLS T5-2;Role T5-2 TimeOut Prezenta Teava OFF;DI;A1;14;O
         DBX140_0 : Bool;
         DBX140_1 : Bool;
         DBX140_2 : Bool;   // 4;ROLLS T5-2;Suma Disj. Th. Vent.Mot. C.Role T5-1 - Declansat;DI;A1;14;M
         DBX140_3 : Bool;   // 4;ROLLS T5-2;TimeOut Cuplare/Decuplare Vent.Mot. C.Role T5-2;DI;A1;14;M;O
         DBX140_4 : Bool;   // 4;ROLLS T5-2;TimeOut Cuplare/Decuplare Alim.Inv. C.Role T5-2;DI;A1;14;M;O;K
         DBX140_5 : Bool;   // 4;ROLLS T5-2;Inverter Mot. C.Role T5-2 - Avarie;DI;A1;14;M;O;K
         DBX140_6 : Bool;
         DBX140_7 : Bool;
         DBX141_0 : Bool;
         DBX141_1 : Bool;
         DBX141_2 : Bool;
         DBX141_3 : Bool;
         DBX141_4 : Bool;
         DBX141_5 : Bool;
         DBX141_6 : Bool;
         DBX141_7 : Bool;
         DBX142_0 : Bool;
         DBX142_1 : Bool;
         DBX142_2 : Bool;
         DBX142_3 : Bool;
         DBX142_4 : Bool;
         DBX142_5 : Bool;
         DBX142_6 : Bool;
         DBX142_7 : Bool;
         DBX143_0 : Bool;
         DBX143_1 : Bool;
         DBX143_2 : Bool;
         DBX143_3 : Bool;
         DBX143_4 : Bool;
         DBX143_5 : Bool;
         DBX143_6 : Bool;
         DBX143_7 : Bool;
         DBX144_0 : Bool;
         DBX144_1 : Bool;
         DBX144_2 : Bool;
         DBX144_3 : Bool;
         DBX144_4 : Bool;
         DBX144_5 : Bool;
         DBX144_6 : Bool;
         DBX144_7 : Bool;
         DBX145_0 : Bool;
         DBX145_1 : Bool;
         DBX145_2 : Bool;
         DBX145_3 : Bool;
         DBX145_4 : Bool;
         DBX145_5 : Bool;
         DBX145_6 : Bool;
         DBX145_7 : Bool;
         DBX146_0 : Bool;   // 4;EXCENTRIC T6;TimeOut Deplasare Inainte Excentric T6;DI;A1;15;M;O;K
         DBX146_1 : Bool;   // 4;EXCENTRIC T6;TimeOut Deplasare Inapoi Excentric T6;DI;A1;15;M;O;K
         DBX146_2 : Bool;   // 4;EXCENTRIC T6;TimeOut Deplasare Excentric T6 in Pozitie;DI;A1;15;M;O;K
         DBX146_3 : Bool;   // 4;EXCENTRIC T6;Disjunctor Termic Mot. Excentric T6 - Declansat;DI;A1;15;M;K
         DBX146_4 : Bool;   // 4;EXCENTRIC T6;Alim. SoftStarter SIKO Excentric T6 - Decuplat;DI;A1;15;M;K
         DBX146_5 : Bool;   // 4;EXCENTRIC T6;Alim. Frana Mot. Excentric T6 - Decuplat;DI;A1;15;M;K
         DBX146_6 : Bool;   // 4;EXCENTRIC T6;Lipsa Tensiune de Comanda Excentric T6;DI;A1;15;M;K
         DBX146_7 : Bool;   // 4;EXCENTRIC T6;SoftStarter SIKO Excentric T6 - Avarie;DI;A1;15;M;O;K
         DBX147_0 : Bool;   // 4;EXCENTRIC T6;Eroare Depozitare Teava pe Pat Racire T6;SQ;A1;15;O
         DBX147_1 : Bool;
         DBX147_2 : Bool;
         DBX147_3 : Bool;
         DBX147_4 : Bool;
         DBX147_5 : Bool;
         DBX147_6 : Bool;
         DBX147_7 : Bool;
         DBX148_0 : Bool;
         DBX148_1 : Bool;
         DBX148_2 : Bool;
         DBX148_3 : Bool;
         DBX148_4 : Bool;
         DBX148_5 : Bool;
         DBX148_6 : Bool;
         DBX148_7 : Bool;
         DBX149_0 : Bool;
         DBX149_1 : Bool;
         DBX149_2 : Bool;
         DBX149_3 : Bool;
         DBX149_4 : Bool;
         DBX149_5 : Bool;
         DBX149_6 : Bool;
         DBX149_7 : Bool;
         DBX150_0 : Bool;   // 4;CHAIN T6;TimeOut Cuplare/Decuplare Alim.Inv. Lant T6;DI;A1;15;M;O;K
         DBX150_1 : Bool;   // 4;CHAIN T6;TimeOut Deplasare Lant T6;DI;A1;15;M;O;K
         DBX150_2 : Bool;   // 4;CHAIN T6;TimeOut Deplasare Lant T6 in pozitia Pas;DI;A1;15;M;O;K
         DBX150_3 : Bool;   // 4;CHAIN T6;TimeOut Cuplare/Decuplare Frana Lant T6;DI;A1;15;M;O;K
         DBX150_4 : Bool;   // 4;CHAIN T6;Sectionator Alim.Inv. Mot. Lant T6 - Decuplat;DI;A1;15;M;K
         DBX150_5 : Bool;   // 4;CHAIN T6;Stop Permisie Cuplare Lant T6 - Actionat;DI;A1;15;M;K
         DBX150_6 : Bool;   // 4;CHAIN T6;Disj. Termic Alim. Vent.Mot. Lant T6 - Declansat;DI;W1;15;M
         DBX150_7 : Bool;   // 4;CHAIN T6;Lipsa Tensiune de Comanda Lant T6;DI;A1;15;M;K
         DBX151_0 : Bool;
         DBX151_1 : Bool;
         DBX151_2 : Bool;   // 4;CHAIN T6;Inverter Mot. Lant T6 - Avarie;DI;A1;15;M;O;K
         DBX151_3 : Bool;   // 4;CHAIN T6;Eroare Depozitare Teava pe Opritor dupa Lant T6;DI;A1;15;O
         DBX151_4 : Bool;   // 4;CHAIN T6;Senzor Incetinire T6 - Avarie (blocat pe "activat");DI;A1;15;M;O;K
         DBX151_5 : Bool;
         DBX151_6 : Bool;
         DBX151_7 : Bool;
         DBX152_0 : Bool;
         DBX152_1 : Bool;
         DBX152_2 : Bool;
         DBX152_3 : Bool;
         DBX152_4 : Bool;
         DBX152_5 : Bool;
         DBX152_6 : Bool;
         DBX152_7 : Bool;
         DBX153_0 : Bool;
         DBX153_1 : Bool;
         DBX153_2 : Bool;
         DBX153_3 : Bool;
         DBX153_4 : Bool;
         DBX153_5 : Bool;
         DBX153_6 : Bool;
         DBX153_7 : Bool;
         DBX154_0 : Bool;   // 4;STOPPER T6;Lipsa Tensiune Alimentare Opritor T6;DI;A1;15;M;K
         DBX154_1 : Bool;   // 4;STOPPER T6;TimeOut Deplasare Opritor T6 in pozitia Sus;DI;A1;15;M
         DBX154_2 : Bool;   // 4;STOPPER T6;TimeOut Deplasare Opritor T6 in pozitia Jos;DI;A1;15;M
         DBX154_3 : Bool;   // 4;STOPPER T6;Eroare Depozitare Teava pe C.Role T6;SQ;A1;15;O
         DBX154_4 : Bool;
         DBX154_5 : Bool;
         DBX154_6 : Bool;
         DBX154_7 : Bool;
         DBX155_0 : Bool;
         DBX155_1 : Bool;
         DBX155_2 : Bool;
         DBX155_3 : Bool;
         DBX155_4 : Bool;
         DBX155_5 : Bool;
         DBX155_6 : Bool;
         DBX155_7 : Bool;
         DBX156_0 : Bool;
         DBX156_1 : Bool;
         DBX156_2 : Bool;
         DBX156_3 : Bool;
         DBX156_4 : Bool;
         DBX156_5 : Bool;
         DBX156_6 : Bool;
         DBX156_7 : Bool;
         DBX157_0 : Bool;
         DBX157_1 : Bool;
         DBX157_2 : Bool;
         DBX157_3 : Bool;
         DBX157_4 : Bool;
         DBX157_5 : Bool;
         DBX157_6 : Bool;
         DBX157_7 : Bool;
         DBX158_0 : Bool;   // 5;ROLLS T6;Suma Disj. Termice Mot. C.Role T6 - Declansat;DI;A1;15;M;K
         DBX158_1 : Bool;   // 5;ROLLS T6;Sectionator Alim.Inv. Mot. C.Role T6 - Decuplat;DI;A1;15;M;K
         DBX158_2 : Bool;   // 5;ROLLS T6;Lipsa Tensiune de Comanda C.Role T6;DI;A1;15;M;K
         DBX158_3 : Bool;   // 5;ROLLS T6;TimeOut Rotire Role C.Role T6;DI;A1;15;M;O;K
         DBX158_4 : Bool;   // 5;ROLLS T6;Disj. Termic Rola Nr.1 C.Role T6 Declansat;DI;W2;15;M
         DBX158_5 : Bool;   // 5;ROLLS T6;Disj. Termic Rola Nr.2 C.Role T6 Declansat;DI;W2;15;M
         DBX158_6 : Bool;   // 5;ROLLS T6;Disj. Termic Rola Nr.3 C.Role T6 Declansat;DI;W2;15;M
         DBX158_7 : Bool;   // 5;ROLLS T6;Disj. Termic Rola Nr.4 C.Role T6 Declansat;DI;W2;15;M
         DBX159_0 : Bool;   // 5;ROLLS T6;Disj. Termic Rola Nr.5 C.Role T6 Declansat;DI;W2;15;M
         DBX159_1 : Bool;   // 5;ROLLS T6;Disj. Termic Rola Nr.6 C.Role T6 Declansat;DI;W2;15;M
         DBX159_2 : Bool;   // 5;ROLLS T6;Disj. Termic Rola Nr.7 C.Role T6 Declansat;DI;W2;15;M
         DBX159_3 : Bool;   // 5;ROLLS T6;Disj. Termic Rola Nr.8 C.Role T6 Declansat;DI;W2;15;M
         DBX159_4 : Bool;   // 5;ROLLS T6;Disj. Termic Rola Nr.9 C.Role T6 Declansat;DI;W2;15;M
         DBX159_5 : Bool;   // 5;ROLLS T6;Disj. Termic Rola Nr.10 C.Role T6 Declansat;DI;W2;15;M
         DBX159_6 : Bool;   // 5;ROLLS T6;Disj. Th. Alim.Vent.Mot. C.Role T6 Declansat;DI;A1;15;M
         DBX159_7 : Bool;   // 5;ROLLS T6;Eroare Encoder C.Role T6;DI;A1;15;M;O;K
         DBX160_0 : Bool;
         DBX160_1 : Bool;   // 5;ROLLS T6;Inverter Mot. C.Role T6 - Avarie;DI;A1;15;M;O;K
         DBX160_2 : Bool;   // 5;ROLLS T6;Suma Disj. Th. Vent.Mot. C.Role T6 - Declansat;DI;A1;15;M
         DBX160_3 : Bool;   // 5;ROLLS T6;TimeOut Cuplare/Decuplare Vent.Mot. C.Role T6;DI;A1;15;M;O
         DBX160_4 : Bool;   // 5;ROLLS T6;TimeOut Cuplare/Decuplare Alim.Inv. C.Role T6;DI;A1;15;M;O;K
         DBX160_5 : Bool;   // 5;ROLLS T6;Role T6 TimeOut LB Masurare Lungime ON;SQ;A1;15;M;O
         DBX160_6 : Bool;   // 5;ROLLS T6;Role T6 TimeOut LB Masurare Lungime OFF;SQ;A1;15;M;O
         DBX160_7 : Bool;   // 5;ROLLS T6;Role T6 TimeOut LB Intrare Cuptor OFF;SQ;A1;15;M;O
         DBX161_0 : Bool;
         DBX161_1 : Bool;
         DBX161_2 : Bool;
         DBX161_3 : Bool;
         DBX161_4 : Bool;
         DBX161_5 : Bool;
         DBX161_6 : Bool;
         DBX161_7 : Bool;
         DBX162_0 : Bool;   // 5;FLIPPER T1-D;Lipsa Tensiune Alimentare Aruncator T1-D;DI;A1;16;M;K
         DBX162_1 : Bool;   // 5;FLIPPER T1-D;TimeOut Deplasare Aruncator T1-D in pozitia Sus;DI;A1;16;M;O
         DBX162_2 : Bool;   // 5;FLIPPER T1-D;TimeOut Deplasare Aruncator T1-D in pozitia Jos;DI;A1;16;M;O
         DBX162_3 : Bool;   // 5;STOPPER T1-D;Disjunctor Termic Opritor T1-D - Declansat;DI;A1;16;M;K
         DBX162_4 : Bool;   // 5;STOPPER T1-D;Sectionator Alimentare Opritor T1-D - Decuplat;DI;A1;16;M;K
         DBX162_5 : Bool;   // 5;STOPPER T1-D;TimeOut Cuplare/Decuplare Contactor Opritor T1D;DI;A1;16;M;O;K
         DBX162_6 : Bool;   // 5;STOPPER T1-D;Eroare Depozitare Teava pe C.Role T1-D;SQ;A1;16;O
         DBX162_7 : Bool;
         DBX163_0 : Bool;
         DBX163_1 : Bool;
         DBX163_2 : Bool;
         DBX163_3 : Bool;
         DBX163_4 : Bool;
         DBX163_5 : Bool;
         DBX163_6 : Bool;
         DBX163_7 : Bool;
         DBX164_0 : Bool;
         DBX164_1 : Bool;
         DBX164_2 : Bool;
         DBX164_3 : Bool;
         DBX164_4 : Bool;
         DBX164_5 : Bool;
         DBX164_6 : Bool;
         DBX164_7 : Bool;
         DBX165_0 : Bool;
         DBX165_1 : Bool;
         DBX165_2 : Bool;
         DBX165_3 : Bool;
         DBX165_4 : Bool;
         DBX165_5 : Bool;
         DBX165_6 : Bool;
         DBX165_7 : Bool;
         DBX166_0 : Bool;   // 5;ROLLS T1-D;Suma Disj. Termice Mot. C.Role T1-D - Declansat;DI;A1;16;M;K
         DBX166_1 : Bool;   // 5;ROLLS T1-D;Sectionator Alim.Inverter C.Role T1-D - Decuplat;DI;A1;16;M;K
         DBX166_2 : Bool;   // 5;ROLLS T1-D;Lipsa Tensiune de Comanda C.Role T1-D;DI;A1;16;M;K
         DBX166_3 : Bool;   // 5;ROLLS T1-D;TimeOut Rotire Role C.Role T1-D;DI;A1;16;M;O;K
         DBX166_4 : Bool;   // 5;ROLLS T1-D;Disj. Termic Rola Nr.1 C.Role T1-D Declansat;DI;W2;16;M
         DBX166_5 : Bool;   // 5;ROLLS T1-D;Disj. Termic Rola Nr.2 C.Role T1-D Declansat;DI;W2;16;M
         DBX166_6 : Bool;   // 5;ROLLS T1-D;Disj. Termic Rola Nr.3 C.Role T1-D Declansat;DI;W2;16;M
         DBX166_7 : Bool;   // 5;ROLLS T1-D;Disj. Termic Rola Nr.4 C.Role T1-D Declansat;DI;W2;16;M
         DBX167_0 : Bool;   // 5;ROLLS T1-D;Disj. Termic Rola Nr.5 C.Role T1-D Declansat;DI;W2;16;M
         DBX167_1 : Bool;   // 5;ROLLS T1-D;Disj. Termic Rola Nr.6 C.Role T1-D Declansat;DI;W2;16;M
         DBX167_2 : Bool;   // 5;ROLLS T1-D;Disj. Termic Rola Nr.7 C.Role T1-D Declansat;DI;W2;16;M
         DBX167_3 : Bool;   // 5;ROLLS T1-D;Disj. Termic Rola Nr.8 C.Role T1-D Declansat;DI;W2;16;M
         DBX167_4 : Bool;   // 5;ROLLS T1-D;Inverter Mot. C.Role T1-D - Avarie;DI;A1;16;M;O;K
         DBX167_5 : Bool;   // 5;ROLLS T1-D;Disjunctor Th. Alim.Vent.Mot.C.Role T1-D-Declansat;DI;A1;16;M
         DBX167_6 : Bool;   // 5;ROLLS T1-D;Eroare Encoder C.Role T1-D;DI;A1;16;M;O;K
         DBX167_7 : Bool;   // 5;ROLLS T1-D;Role T1-D TimeOut LB Masurare Lungime ON;SQ;A1;16;M
         DBX168_0 : Bool;   // 5;ROLLS T1-D;Role T1-D TimeOut LB Masurare Lungime OFF;SQ;A1;16;M
         DBX168_1 : Bool;
         DBX168_2 : Bool;   // 5;ROLLS T1-D;Suma Disj. Termice Vent.Mot.C.Role T1-D-Declansa;DI;A1;16;M
         DBX168_3 : Bool;   // 5;ROLLS T1-D;TimeOut Cuplare/Decuplare Vent.Mot. C.Role T1-D;DI;A1;16;M;O
         DBX168_4 : Bool;   // 5;ROLLS T1-D;TimeOut Cuplare Alim.Inverter C.Role T1-D;DI;A1;16;M;O;K
         DBX168_5 : Bool;
         DBX168_6 : Bool;
         DBX168_7 : Bool;
         DBX169_0 : Bool;
         DBX169_1 : Bool;
         DBX169_2 : Bool;
         DBX169_3 : Bool;
         DBX169_4 : Bool;
         DBX169_5 : Bool;
         DBX169_6 : Bool;
         DBX169_7 : Bool;
         DBX170_0 : Bool;
         DBX170_1 : Bool;
         DBX170_2 : Bool;
         DBX170_3 : Bool;
         DBX170_4 : Bool;
         DBX170_5 : Bool;
         DBX170_6 : Bool;
         DBX170_7 : Bool;
         DBX171_0 : Bool;
         DBX171_1 : Bool;
         DBX171_2 : Bool;
         DBX171_3 : Bool;
         DBX171_4 : Bool;
         DBX171_5 : Bool;
         DBX171_6 : Bool;
         DBX171_7 : Bool;
         DBX172_0 : Bool;
         DBX172_1 : Bool;
         DBX172_2 : Bool;
         DBX172_3 : Bool;
         DBX172_4 : Bool;
         DBX172_5 : Bool;
         DBX172_6 : Bool;
         DBX172_7 : Bool;
         DBX173_0 : Bool;
         DBX173_1 : Bool;
         DBX173_2 : Bool;
         DBX173_3 : Bool;
         DBX173_4 : Bool;
         DBX173_5 : Bool;
         DBX173_6 : Bool;
         DBX173_7 : Bool;
         DBX174_0 : Bool;   // 8;ROLLS T7;Suma Disj. Termice Mot. C.Role T7 - Declansat;DI;A1;21;M;K
         DBX174_1 : Bool;   // 8;ROLLS T7;Sectionator Alim.Inv. Mot. C.Role T7 - Decuplat;DI;A1;21;M;K
         DBX174_2 : Bool;   // 8;ROLLS T7;Lipsa Tensiune de Comanda C.Role T7;DI;A1;21;M;K
         DBX174_3 : Bool;   // 8;ROLLS T7;TimeOut Rotire Role C.Role T7;DI;A1;21;M;O;K
         DBX174_4 : Bool;   // 8;ROLLS T7;Disj. Termic Rola Nr.1 C.Role T7 Declansat;DI;W2;21;M
         DBX174_5 : Bool;   // 8;ROLLS T7;Disj. Termic Rola Nr.2 C.Role T7 Declansat;DI;W2;21;M
         DBX174_6 : Bool;   // 8;ROLLS T7;Disj. Termic Rola Nr.3 C.Role T7 Declansat;DI;W2;21;M
         DBX174_7 : Bool;   // 8;ROLLS T7;Disj. Termic Rola Nr.4 C.Role T7 Declansat;DI;W2;21;M
         DBX175_0 : Bool;   // 8;ROLLS T7;Disj. Termic Rola Nr.5 C.Role T7 Declansat;DI;W2;21;M
         DBX175_1 : Bool;   // 8;ROLLS T7;Disj. Termic Rola Nr.6 C.Role T7 Declansat;DI;W2;21;M
         DBX175_2 : Bool;   // 8;ROLLS T7;Disj. Termic Rola Nr.7 C.Role T7 Declansat;DI;W2;21;M
         DBX175_3 : Bool;   // 8;ROLLS T7;Disj. Termic Rola Nr.8 C.Role T7 Declansat;DI;W2;21;M
         DBX175_4 : Bool;   // 8;ROLLS T7;Disj. Termic Rola Nr.9 C.Role T7 Declansat;DI;W2;21;M
         DBX175_5 : Bool;   // 8;ROLLS T7;Disj. Termic Rola Nr.10 C.Role T7 Declansat;DI;W2;21;M
         DBX175_6 : Bool;   // 8;ROLLS T7;Inverter Mot. C.Role T7 Avarie;DI;A1;21;M;O;K
         DBX175_7 : Bool;
         DBX176_0 : Bool;
         DBX176_1 : Bool;
         DBX176_2 : Bool;   // 8;ROLLS T7;Suma Disj. Th. Vent.Mot. C.Role T7 - Declansat;DI;A1;21;M
         DBX176_3 : Bool;   // 8;ROLLS T7;TimeOut Cuplare/Decuplare Vent.Mot. C.Role T7;DI;A1;21;M;O
         DBX176_4 : Bool;   // 8;ROLLS T7;TimeOut Cuplare/Decuplare Alim.Inv. C.Role T7;DI;A1;21;M;O;K
         DBX176_5 : Bool;   // 8;ROLLS T7;Disj. Th. Alim.Vent.Mot. C.Role T7 - Declansat;DI;A1;21;M
         DBX176_6 : Bool;   // 8;ROLLS T7;Role T7 TimeOut LB Iesire Cuptor ON;SQ;A1;21;O
         DBX176_7 : Bool;   // 8;ROLLS T7;Role T7 TimeOut LB Iesire Cuptor OFF;SQ;A1;21;O
         DBX177_0 : Bool;   // 8;ROLLS T7;Role T7 TimeOut LB Viteza Redusa ON;SQ;A1;21;O
         DBX177_1 : Bool;   // 8;ROLLS T7;Role T7 TimeOut LB Pozitionare Teava;SQ;A1;21;O
         DBX177_2 : Bool;
         DBX177_3 : Bool;
         DBX177_4 : Bool;
         DBX177_5 : Bool;
         DBX177_6 : Bool;
         DBX177_7 : Bool;
         DBX178_0 : Bool;   // 8;FLIPPER T7;Lipsa Tensiune Alimentare Aruncator T7;DI;A1;21;M;K
         DBX178_1 : Bool;   // 8;FLIPPER T7;TimeOut Deplasare Aruncator T7 in pozitia Sus;DI;A1;21;M;O
         DBX178_2 : Bool;   // 8;FLIPPER T7;TimeOut Deplasare Aruncator T7 in pozitia Jos;DI;A1;21;M;O
         DBX178_3 : Bool;   // 8;FLIPPER T7;Eroare Depoz. Teava pe Poz.PreluareExcentric 1 T7;DI;A1;21;O
         DBX178_4 : Bool;
         DBX178_5 : Bool;
         DBX178_6 : Bool;
         DBX178_7 : Bool;
         DBX179_0 : Bool;
         DBX179_1 : Bool;
         DBX179_2 : Bool;
         DBX179_3 : Bool;
         DBX179_4 : Bool;
         DBX179_5 : Bool;
         DBX179_6 : Bool;
         DBX179_7 : Bool;
         DBX180_0 : Bool;
         DBX180_1 : Bool;
         DBX180_2 : Bool;
         DBX180_3 : Bool;
         DBX180_4 : Bool;
         DBX180_5 : Bool;
         DBX180_6 : Bool;
         DBX180_7 : Bool;
         DBX181_0 : Bool;
         DBX181_1 : Bool;
         DBX181_2 : Bool;
         DBX181_3 : Bool;
         DBX181_4 : Bool;
         DBX181_5 : Bool;
         DBX181_6 : Bool;
         DBX181_7 : Bool;
         DBX182_0 : Bool;   // 8;EXC.1 T7;TimeOut Deplasare Inainte Excentric 1 C.Role T7;DI;A1;21;M;O
         DBX182_1 : Bool;   // 8;EXC.1 T7;TimeOut Deplasare Inapoi Excentric 1 C.Role T7;DI;A1;21;M;O
         DBX182_2 : Bool;   // 8;EXC.1 T7;TimeOut Deplasare Excentric 1 C.Role T7 in Pozitie;DI;A1;21;M;O
         DBX182_3 : Bool;   // 8;EXC.1 T7;Disjunc. Termic Mot. Excentric 1C.Role T7-Declansat;DI;A1;21;M;K
         DBX182_4 : Bool;   // 8;EXC.1 T7;Alim. SoftStart.SIKO Excentric 1 C.Role T7-Decuplat;DI;A1;21;M;K
         DBX182_5 : Bool;   // 8;EXC.1 T7;Alim. Frana Mot. Excentric 1 C.Role T7 - Decuplat;DI;A1;21;M;K
         DBX182_6 : Bool;   // 8;EXC.1 T7;Lipsa Tensiune de Comanda Excentric 1 C.Role T7;DI;A1;21;M;K
         DBX182_7 : Bool;   // 8;EXC.1 T7;SoftStarter SIKO Excentric 1 C.Role T7 - Avarie;DI;A1;21;M;O;K
         DBX183_0 : Bool;
         DBX183_1 : Bool;
         DBX183_2 : Bool;
         DBX183_3 : Bool;
         DBX183_4 : Bool;
         DBX183_5 : Bool;
         DBX183_6 : Bool;
         DBX183_7 : Bool;
         DBX184_0 : Bool;
         DBX184_1 : Bool;
         DBX184_2 : Bool;
         DBX184_3 : Bool;
         DBX184_4 : Bool;
         DBX184_5 : Bool;
         DBX184_6 : Bool;
         DBX184_7 : Bool;
         DBX185_0 : Bool;
         DBX185_1 : Bool;
         DBX185_2 : Bool;
         DBX185_3 : Bool;
         DBX185_4 : Bool;
         DBX185_5 : Bool;
         DBX185_6 : Bool;
         DBX185_7 : Bool;
         DBX186_0 : Bool;   // 8;EXC.2 T7;TimeOut Deplasare Inainte Excentric 2 C.Role T7;DI;A1;21;M;O
         DBX186_1 : Bool;   // 8;EXC.2 T7;TimeOut Deplasare Inapoi Excentric 2 C.Role T7;DI;A1;21;M;O
         DBX186_2 : Bool;   // 8;EXC.2 T7;TimeOut Deplasare Excentric 2 C.Role T7 in Pozitie;DI;A1;21;M;O
         DBX186_3 : Bool;   // 8;EXC.2 T7;Disjunc. Termic Mot. Excentric 2C.Role T7-Declansat;DI;A1;21;M;K
         DBX186_4 : Bool;   // 8;EXC.2 T7;Alim. SoftStart. SIKO Excentric 2C.Role T7-Decuplat;DI;A1;21;M;K
         DBX186_5 : Bool;   // 8;EXC.2 T7;Alim. Frana Mot. Excentric 2 C.Role T7 - Decuplat;DI;A1;21;M;K
         DBX186_6 : Bool;   // 8;EXC.2 T7;Lipsa Tensiune de Comanda Excentric 2 C.Role T7;DI;A1;21;M;K
         DBX186_7 : Bool;   // 8;EXC.2 T7;SoftStarter SIKO Excentric 2 C.Role T7 - Avarie;DI;A1;21;M;O;K
         DBX187_0 : Bool;   // 8;EXC.2 T7;Eroare Depozitare Teava pe Poz. Asteptare la SUTTON;SQ;A1;21;O
         DBX187_1 : Bool;   // 8;EXC.2 T7;Lipsa racire role Lazzarri;DI;A2;21;O;K
         DBX187_2 : Bool;
         DBX187_3 : Bool;
         DBX187_4 : Bool;
         DBX187_5 : Bool;
         DBX187_6 : Bool;
         DBX187_7 : Bool;
         DBX188_0 : Bool;
         DBX188_1 : Bool;
         DBX188_2 : Bool;
         DBX188_3 : Bool;
         DBX188_4 : Bool;
         DBX188_5 : Bool;
         DBX188_6 : Bool;
         DBX188_7 : Bool;
         DBX189_0 : Bool;
         DBX189_1 : Bool;
         DBX189_2 : Bool;
         DBX189_3 : Bool;
         DBX189_4 : Bool;
         DBX189_5 : Bool;
         DBX189_6 : Bool;
         DBX189_7 : Bool;
         DBX190_0 : Bool;
         DBX190_1 : Bool;
         DBX190_2 : Bool;
         DBX190_3 : Bool;
         DBX190_4 : Bool;
         DBX190_5 : Bool;
         DBX190_6 : Bool;
         DBX190_7 : Bool;
         DBX191_0 : Bool;
         DBX191_1 : Bool;
         DBX191_2 : Bool;
         DBX191_3 : Bool;
         DBX191_4 : Bool;
         DBX191_5 : Bool;
         DBX191_6 : Bool;
         DBX191_7 : Bool;
         DBX192_0 : Bool;
         DBX192_1 : Bool;
         DBX192_2 : Bool;
         DBX192_3 : Bool;
         DBX192_4 : Bool;
         DBX192_5 : Bool;
         DBX192_6 : Bool;
         DBX192_7 : Bool;
         DBX193_0 : Bool;
         DBX193_1 : Bool;
         DBX193_2 : Bool;
         DBX193_3 : Bool;
         DBX193_4 : Bool;
         DBX193_5 : Bool;
         DBX193_6 : Bool;
         DBX193_7 : Bool;
         DBX194_0 : Bool;   // 9;EXCENTRIC-1 T7A;TimeOut Deplasare Inainte Excentric 1 Lant T7A;DI;A1;23;M;O;K
         DBX194_1 : Bool;   // 9;EXCENTRIC-1 T7A;TimeOut Deplasare Inapoi Excentric 1 Lant T7-A;DI;A1;23;M;O;K
         DBX194_2 : Bool;   // 9;EXCENTRIC-1 T7A;TimeOut Deplasare Excentr. 1 Lant T7-A Pozitie.;DI;A1;23;M;O
         DBX194_3 : Bool;   // 9;EXCENTRIC-1 T7A;Disj. Th. Mot. Excentric 1 Lant T7-A-Declansat;DI;A2;23;M;K
         DBX194_4 : Bool;   // 9;EXCENTRIC-1 T7A;Alim. SoftStart Excentric 1 Lant T7-A-Decuplat;DI;A2;23;M;K
         DBX194_5 : Bool;   // 9;EXCENTRIC-1 T7A;Alim. Frana Mot. Excentric 1 Lant T7A-Decuplat;DI;A2;23;M;K
         DBX194_6 : Bool;   // 9;EXCENTRIC-1 T7A;Lipsa Tensiune de Comanda Excentric 1 Lant T7A;DI;A1;23;M;K
         DBX194_7 : Bool;   // 9;EXCENTRIC-1 T7A;SoftStarter SIKO Excentric 1 Lant T7A - Avarie;DI;A1;23;M;O;K
         DBX195_0 : Bool;   // 9;EXCENTRIC-1 T7A;Eroare Depozitare Teava pe Lant T7-A;SQ;A1;23;O
         DBX195_1 : Bool;
         DBX195_2 : Bool;
         DBX195_3 : Bool;
         DBX195_4 : Bool;
         DBX195_5 : Bool;
         DBX195_6 : Bool;
         DBX195_7 : Bool;
         DBX196_0 : Bool;
         DBX196_1 : Bool;
         DBX196_2 : Bool;
         DBX196_3 : Bool;
         DBX196_4 : Bool;
         DBX196_5 : Bool;
         DBX196_6 : Bool;
         DBX196_7 : Bool;
         DBX197_0 : Bool;
         DBX197_1 : Bool;
         DBX197_2 : Bool;
         DBX197_3 : Bool;
         DBX197_4 : Bool;
         DBX197_5 : Bool;
         DBX197_6 : Bool;
         DBX197_7 : Bool;
         DBX198_0 : Bool;
         DBX198_1 : Bool;
         DBX198_2 : Bool;   // 9;CHAIN T7A;Stop Permisie Cuplare Lant T7-A - Actionat;DI;A1;23;M;K
         DBX198_3 : Bool;   // 9;CHAIN T7A;TimeOut Cuplare/Decuplare Alim.Inv. Lant T7-A;DI;A1;23;M;O;K
         DBX198_4 : Bool;   // 9;CHAIN T7A;Lipsa Tensiune de Comanda Lant T7-A;DI;A1;23;M;K
         DBX198_5 : Bool;   // 9;CHAIN T7A;Sectionator Alim.Inv. Mot. Lant T7-A - Decuplat;DI;A1;23;M;K
         DBX198_6 : Bool;   // 9;CHAIN T7A;Disjunctor Thermic Mot. Lant T7-A - Declansat;DI;A1;23;M;K
         DBX198_7 : Bool;   // 9;CHAIN T7A;Inverter Mot. Lant T7-A - Avarie;DI;A1;23;M;O;K
         DBX199_0 : Bool;   // 9;CHAIN T7A SPIN;TimeOut Cuplare/Decup Alim.Inv. LantRost. T7-A;DI;A1;23;M;O;K
         DBX199_1 : Bool;   // 9;CHAIN T7A SPIN;Sectionator Alim.Inv Mot. LantRost T7A-Decuplat;DI;A1;23;M;K
         DBX199_2 : Bool;   // 9;CHAIN T7A SPIN;Disjunctor Termic Mot. LantRost. T7-A-Declansat;DI;A1;23;M;K
         DBX199_3 : Bool;   // 9;CHAIN T7A;TimeOut Deplasare Lant T7-A in pozitia Pas;DI;A1;23;M;O;K
         DBX199_4 : Bool;   // 9;CHAIN T7A SPIN;Inverter Mot. Lant Rost. T7-A - Avarie;DI;A2;23;M;O;K
         DBX199_5 : Bool;
         DBX199_6 : Bool;
         DBX199_7 : Bool;
         DBX200_0 : Bool;
         DBX200_1 : Bool;
         DBX200_2 : Bool;
         DBX200_3 : Bool;
         DBX200_4 : Bool;
         DBX200_5 : Bool;
         DBX200_6 : Bool;
         DBX200_7 : Bool;
         DBX201_0 : Bool;
         DBX201_1 : Bool;
         DBX201_2 : Bool;
         DBX201_3 : Bool;
         DBX201_4 : Bool;
         DBX201_5 : Bool;
         DBX201_6 : Bool;
         DBX201_7 : Bool;
         DBX202_0 : Bool;   // 9;EXCENTRIC-2 T7A;TimeOut Deplasare Inainte Excentric2 Lant T7-A;DI;A1;23;M;O;K
         DBX202_1 : Bool;   // 9;EXCENTRIC-2 T7A;TimeOut Deplasare Inapoi Excentric 2 Lant T7-A;DI;A1;23;M;O;K
         DBX202_2 : Bool;   // 9;EXCENTRIC-2 T7A;TimeOut Deplasare Excentric 2 Lant T7-A Pozitie;DI;A1;23;O;M
         DBX202_3 : Bool;   // 9;EXCENTRIC-2 T7A;Disj. Th. Mot. Excentric 2 Lant T7-A-Declansat;DI;A2;23;M;K
         DBX202_4 : Bool;   // 9;EXCENTRIC-2 T7A;Alim. SoftStart Excentric 2 Lant T7-A-Decuplat;DI;A2;23;M;K
         DBX202_5 : Bool;   // 9;EXCENTRIC-2 T7A;Alim. Frana Mot. Excentric 2 Lant T7A-Decuplat;DI;A2;23;M;K
         DBX202_6 : Bool;   // 9;EXCENTRIC-2 T7A;Lipsa Tensiune de Comanda Excentric 2 Lant T7A;DI;A1;23;M;K
         DBX202_7 : Bool;   // 9;EXCENTRIC-2 T7A;SoftStarter SIKO Excentric 2 Lant T7A - Avarie;DI;A1;23;M;O;K
         DBX203_0 : Bool;   // 9;EXCENTRIC-2 T7A;Eroare Depozitare Teava pe C.Role T7-A;SQ;A1;23;O
         DBX203_1 : Bool;
         DBX203_2 : Bool;
         DBX203_3 : Bool;
         DBX203_4 : Bool;
         DBX203_5 : Bool;
         DBX203_6 : Bool;
         DBX203_7 : Bool;
         DBX204_0 : Bool;
         DBX204_1 : Bool;
         DBX204_2 : Bool;
         DBX204_3 : Bool;
         DBX204_4 : Bool;
         DBX204_5 : Bool;
         DBX204_6 : Bool;
         DBX204_7 : Bool;
         DBX205_0 : Bool;
         DBX205_1 : Bool;
         DBX205_2 : Bool;
         DBX205_3 : Bool;
         DBX205_4 : Bool;
         DBX205_5 : Bool;
         DBX205_6 : Bool;
         DBX205_7 : Bool;
         DBX206_0 : Bool;   // 9;ROLE T7A;TimeOut Rotire Role C.Role T7-A;DI;A1;23;M;O
         DBX206_1 : Bool;   // 9;ROLE T7A;Lipsa Tensiune de Comanda C.Role T7-A;DI;A1;23;M;K
         DBX206_2 : Bool;   // 9;ROLE T7A;Sectionator Alim.Inv. Mot. C.Role T7-A Decuplat;DI;A2;23;M;K
         DBX206_3 : Bool;   // 9;ROLE T7A;Suma Disj. Th. Vent.Mot. C.Role T7-A Declansat;DI;A1;23;M
         DBX206_4 : Bool;   // 9;ROLE T7A;TimeOut Cuplare/Decuplare Vent.Mot. C.Role T7-A;DI;A1;23;M;O
         DBX206_5 : Bool;   // 9;ROLE T7A;TimeOut Cuplare/Decuplare Alim.Inv. C.Role T7-A;DI;A1;23;M;O;K
         DBX206_6 : Bool;   // 9;ROLE T7A;Role T7-A TimeOut Teava pe Calea Cu Role T7-B;SQ;A1;23;O
         DBX206_7 : Bool;   // 9;ROLE T7A;Role T7-A TimeOut Teava OFF;SQ;A1;23;O
         DBX207_0 : Bool;
         DBX207_1 : Bool;
         DBX207_2 : Bool;
         DBX207_3 : Bool;
         DBX207_4 : Bool;
         DBX207_5 : Bool;
         DBX207_6 : Bool;   // 9;ROLE T7A;Suma Disj. Termice Mot. C.Role T7-A Declansat;DI;A1;23;M;K
         DBX207_7 : Bool;   // 9;ROLE T7A;Inverter Mot. C.Role T7-A Avarie;DI;A2;23;M;O;K
         DBX208_0 : Bool;   // 9;MARCATOR;24 VDC power supply fault;DI;A2;23;O;K
         DBX208_1 : Bool;   // 9;MARCATOR;Robot controller Profinet connection Fault;DI;A2;23;O;K
         DBX208_2 : Bool;   // 9;MARCATOR;Laser sensor (IL-600) Profinet connection Fault;DI;A2;23;O;K
         DBX208_3 : Bool;   // 9;MARCATOR;Datamatrix Reader (Cognex) Profinet connection Fault;DI;A2;23;O;K
         DBX208_4 : Bool;   // 9;MARCATOR;Electric Lock (Fortress) Profinet connection Fault;DI;A2;23;O;K
         DBX208_5 : Bool;   // 9;MARCATOR;REAJET system power supply Fault;DI;A2;23;O;K
         DBX208_6 : Bool;   // 9;MARCATOR;Paint Cabinet Fan power supply Fault;DI;A2;23;O;K
         DBX208_7 : Bool;   // 9;MARCATOR;Smoke Extractor power supply Fault;DI;A2;23;O;K
         DBX209_0 : Bool;   // 9;MARCATOR;Pipe position detection Encoder Fault signalization;DI;A2;23;O;K
         DBX209_1 : Bool;   // 9;MARCATOR;Pipe presence detect Lasersens(LR-TB2000)vitality Fault;DI;A2;23;O;K
         DBX209_2 : Bool;   // 9;MARCATOR;Pipe diam detect Lasersens(IL-600)Fault signalization;DI;A2;23;O;K
         DBX209_3 : Bool;   // 9;MARCATOR;Compressed air low pressure;DI;W2;23;O;K
         DBX209_4 : Bool;   // 9;MARCATOR;Fumes Extractor filter clogged;DI;W2;23;O;K
         DBX209_5 : Bool;   // 9;MARCATOR;Black Paint paint low level;DI;W2;23;O;K
         DBX209_6 : Bool;   // 9;MARCATOR;Black Paint solvent low level;DI;W2;23;O;K
         DBX209_7 : Bool;   // 9;MARCATOR;REAJET Solvent empty (from Paint Cabinet);DI;W2;23;O;K
         DBX210_0 : Bool;   // 9;MARCATOR;REAJET Ink low level (from Ink Device);DI;W2;23;O;K
         DBX210_1 : Bool;   // 9;MARCATOR;REAJET controller not Ready;DI;A2;23;O;K
         DBX210_2 : Bool;   // 9;MARCATOR;REAJET controller Error;DI;A2;23;O;K
         DBX210_3 : Bool;   // 9;MARCATOR;one or more presets wrong;DI;A2;23;O;K
         DBX210_4 : Bool;   // 9;MARCATOR;Pipe Diameter set is out of range;DI;A2;23;O;K
         DBX210_5 : Bool;   // 9;MARCATOR;Pipe Length set is out of range;DI;A2;23;O;K
         DBX210_6 : Bool;   // 9;MARCATOR;1=marking cycle aborted, pipe diam detected is diff;DI;A2;23;O;K
         DBX210_7 : Bool;   // 9;MARCATOR;1<= Datamatrix not recognized on Pipe after marking;DI;A2;23;O;K
         DBX211_0 : Bool;   // 9;MARCATOR;all Datamatrix not recognized on Pipe after marking;DI;A2;23;O;K
         DBX211_1 : Bool;   // 9;MARCATOR;Pipe presence lost before marking cycle completion;DI;A2;23;O;K
         DBX211_2 : Bool;   // 9;MARCATOR;Robot Emergency ON;DI;A2;23;O;K
         DBX211_3 : Bool;   // 9;MARCATOR;1 = AUTO mode on but Motors are off;DI;A2;23;O;K
         DBX211_4 : Bool;   // 9;MARCATOR;1 = Robot controller system failure;DI;A2;23;O;K
         DBX211_5 : Bool;   // 9;MARCATOR;1 = collision has occurred;DI;A2;23;O;K
         DBX211_6 : Bool;   // 9;MARCATOR;1 = max number of collisions reached;DI;A2;23;O;K
         DBX211_7 : Bool;   // 9;MARCATOR;1=cycle aborted(activ WHEN robot generates self abort);DI;A2;23;O;K
         DBX212_0 : Bool;   // 9;MARCATOR;1 = cycle start but robot not home position;DI;A2;23;O;K
         DBX212_1 : Bool;   // 9;MARCATOR;1 = the batteries of the robot are low;DI;W2;23;O;K
         DBX212_2 : Bool;   // 9;MARCATOR;1 = power supply has encountered a fault;DI;A2;23;O;K
         DBX212_3 : Bool;   // 9;MARCATOR;Marking cycle timeout;DI;A2;23;O;K
         DBX212_4 : Bool;   // 9;MARCATOR;1 = presets are wrong;DI;A2;23;O;K
         DBX212_5 : Bool;   // 9;MARCATOR;1 = the speed set is outrange;DI;A2;23;O;K
         DBX212_6 : Bool;   // 9;MARCATOR;1 = Emergency Stop Alarm;DI;A2;23;O;K
         DBX212_7 : Bool;   // 9;MARCATOR;1 = Auto Stop Alarm;DI;A2;23;O;K
         DBX213_0 : Bool;   // 9;MARCATOR;1 = Main Emergency Stop;DI;A2;23;O;K
         DBX213_1 : Bool;   // 9;MARCATOR;Mastering Test cycle is requested by the Robot;DI;A2;23;O;K
         DBX213_2 : Bool;   // 9;MARCATOR;Brake Test cycle is requested by the Robot;DI;A2;23;O;K
         DBX213_3 : Bool;   // 9;MARCATOR;The previous Mastering Test cycle completed with error;DI;A2;23;O;K
         DBX213_4 : Bool;   // 9;MARCATOR;The previous Brake Test cycle completed with error;DI;A2;23;O;K
         DBX213_5 : Bool;   // 9;MARCATOR;Communication Error With Level 2(UNMARKED PIPE);DI;A2;23;O;K
         DBX213_6 : Bool;
         DBX213_7 : Bool;
         DBX214_0 : Bool;
         DBX214_1 : Bool;
         DBX214_2 : Bool;
         DBX214_3 : Bool;
         DBX214_4 : Bool;
         DBX214_5 : Bool;
         DBX214_6 : Bool;
         DBX214_7 : Bool;
         DBX215_0 : Bool;
         DBX215_1 : Bool;
         DBX215_2 : Bool;
         DBX215_3 : Bool;
         DBX215_4 : Bool;
         DBX215_5 : Bool;
         DBX215_6 : Bool;
         DBX215_7 : Bool;
         DBX216_0 : Bool;
         DBX216_1 : Bool;
         DBX216_2 : Bool;
         DBX216_3 : Bool;
         DBX216_4 : Bool;
         DBX216_5 : Bool;
         DBX216_6 : Bool;
         DBX216_7 : Bool;
         DBX217_0 : Bool;
         DBX217_1 : Bool;
         DBX217_2 : Bool;
         DBX217_3 : Bool;
         DBX217_4 : Bool;
         DBX217_5 : Bool;
         DBX217_6 : Bool;
         DBX217_7 : Bool;
         DBX218_0 : Bool;   // 9;ROLE T7B;TimeOut Rotire Role C.Role T7-B;DI;A1;26;M;O
         DBX218_1 : Bool;   // 9;ROLE T7B;Lipsa Tensiune de Comanda C.Role T7-B;DI;A1;26;M;K
         DBX218_2 : Bool;   // 9;ROLE T7B;Sectionator Alim.Inv. Mot. C.Role T7-B - Decuplat;DI;A2;26;M;K
         DBX218_3 : Bool;   // 9;ROLE T7B;Suma Disj. Th. Vent.Mot. C.Role T7-B - Declansat;DI;A1;26;M
         DBX218_4 : Bool;   // 9;ROLE T7B;TimeOut Cuplare/Decuplare Vent.Mot. C.Role T7-B;DI;A1;26;M;O
         DBX218_5 : Bool;   // 9;ROLE T7B;TimeOut Cuplare/Decuplare Alim.Inv. C.Role T7-B;DI;A1;26;M;O;K
         DBX218_6 : Bool;   // 9;ROLE T7B;Role T7-B TimeOut Prezenta Teava;SQ;A1;26;O
         DBX218_7 : Bool;   // 9;ROLE T7B;Role T7-B TimeOut Prezenta Teava Viteza Redusa;SQ;A1;26;O
         DBX219_0 : Bool;   // 9;ROLE T7B;Role T7-B TimeOut Pozitionare Teava;SQ;A1;26;O
         DBX219_1 : Bool;   // 9;ROLE T7B;Role T7-B TimeOut Teava Prezenta pe Calea cu Role T7-C;SQ;A1;26;O
         DBX219_2 : Bool;   // 9;ROLE T7B;Role T7-B TimeOut Teava OFF;SQ;A1;26;O
         DBX219_3 : Bool;   // 9;ROLE T7B;Role T7-B TimeOut Pozitionare Teava;SQ;A1;26;O
         DBX219_4 : Bool;
         DBX219_5 : Bool;
         DBX219_6 : Bool;   // 9;ROLE T7B;Suma Disj. Termice Mot. C.Role T7-B - Declansat;DI;A1;26;M;K
         DBX219_7 : Bool;   // 9;ROLE T7B;Inverter Mot. C.Role T7-B - Avarie;DI;A2;26;M;O;K
         DBX220_0 : Bool;
         DBX220_1 : Bool;
         DBX220_2 : Bool;
         DBX220_3 : Bool;
         DBX220_4 : Bool;
         DBX220_5 : Bool;
         DBX220_6 : Bool;
         DBX220_7 : Bool;
         DBX221_0 : Bool;
         DBX221_1 : Bool;
         DBX221_2 : Bool;
         DBX221_3 : Bool;
         DBX221_4 : Bool;
         DBX221_5 : Bool;
         DBX221_6 : Bool;
         DBX221_7 : Bool;
         DBX222_0 : Bool;   // 9;FLIPPER1 T7B;Lipsa Tensiune Alimentare Aruncator 1 T7-B;DI;A1;26;M;K
         DBX222_1 : Bool;   // 9;FLIPPER1 T7B;TimeOut Deplasare Aruncator 1 T7-B in pozitia Sus;DI;A1;26;M;O
         DBX222_2 : Bool;   // 9;FLIPPER1 T7B;TimeOut Deplasare Aruncator 1 T7-B in pozitia Jos;DI;A1;26;M;O
         DBX222_3 : Bool;   // 9;FLIPPER1 T7B;Eroare Depozitare Teava pe Lant T7-B;SQ;A1;26;O
         DBX222_4 : Bool;
         DBX222_5 : Bool;
